// TwinCAT 3 PLC project Test_Projekt
// ProgramVersion: 3.1.4026.14
// libraries:
//   Tc2_Standard, * (Beckhoff Automation GmbH)
//   Tc2_System, * (Beckhoff Automation GmbH)
//   Tc2_Utilities, * (Beckhoff Automation GmbH)
//   Tc3_Module, * (Beckhoff Automation GmbH)
// project tree:
//   DUTs/Enums/ E_CAN_Object_Test_Error_Bits.TcDUT, E_Controlmode.TcDUT, E_Controlword_Bits.TcDUT, E_Homing_mode.TcDUT, E_LoggerState.TcDUT, E_Mode_of_operation.TcDUT, E_Test_step.TcDUT, E_Statemachine_State.TcDUT, E_Statemachine_Transition_Controlword.TcDUT, E_Statusword_Bits.TcDUT, E_SubElement_Types.TcDUT, J_E_Stop_Modes.TcDUT, J_E_Test_Ranking.TcDUT
//   DUTs/Structs/ ST_CAN_Object.TcDUT, ST_Homing_parameters.TcDUT, ST_Manufacturer_label.TcDUT, ST_Profile_velocity_parameters.TcDUT, ST_Statemachine_State.TcDUT, ST_Velocity_parameters.TcDUT
//   GVLs/ DS301_Object_List.TcGVL, DS302_Object_List.TcGVL, DS402_Object_List.TcGVL, GLB.TcGVL, Manufacturer_Label_Objects.TcGVL, Manufacturer_specific_Object_List.TcGVL, PDO.TcGVL
//   / PlcTask.TcTTO
//   POUs/ CAN_Object_Testing.TcPOU, Encoder_Alignment.TcPOU, Homing_Mode.TcPOU, J_Stop_Testing_SM.TcPOU, Velocity_Mode.TcPOU, MAIN.TcPOU, GET_STATE.TcPOU, Profile_Position_Mode.TcPOU, CONTROLWORD_STATE_CHANGE.TcPOU, Profile_Velocity_Mode.TcPOU, WRITE_Manufacturer_label.TcPOU, READ_Manufacturer_label.TcPOU
//   POUs/FB/Basic/ FB_NMT_WRITE.TcPOU, FB_SDO_READ.TcPOU, FB_SDO_READ_REAL.TcPOU, FB_SDO_WRITE.TcPOU, FB_SDO_WRITE_REAL.TcPOU
//   POUs/FB/ FB_DS402_Object_Testing.TcPOU, FB_Logger.TcPOU, FB_Object_List_Testing.TcPOU, FB_Object_Testing.TcPOU, FB_Sequenz_Testing.TcPOU
//   POUs/FUN/ DWORD_TO_BYTE_ARRAY.TcPOU, Get_Vel_RPM.TcPOU, J_Make_Message.TcPOU
// real-time tasks:
//   TASK PlcTask: cycle T#10ms, priority 20, ADS port 350
// I/O:
//   DEVICE Gerät 1 (EtherCAT), AmsNetId 5.156.6.243.2.1
//     Klemme 1 (EK1200) [EK1200-5000 EtherCAT Netzteil (2A E-Bus)]
//       Klemme 2 (EL1859) [EL1859 8K. Dig. Eingang 24V, 3ms, 8K. Dig. Ausgang 24V, 0.5A]
//       Klemme 3 (EL6751) [EL6751 CANopen Master]
//       Klemme 4 (EK1110) [EK1110 EtherCAT-Verlängerung]
//   DEVICE Gerät 3 (NOV-DP-RAM)
//   DEVICE Gerät 2 (EL6751), AmsNetId 5.156.6.243.3.1
//     Box 5 (CANopen Node)
// variable links:
//   Test_Projekt/Test_Projekt Instance <-> Device 1 (EtherCAT)/Term 1 (EK1200)/Term 2 (EL1859)
//     PlcTask Inputs/MAIN.bTaster{1..8} <-> Channel {1..8}/Input  (8 links)
//     PlcTask Outputs/MAIN.Stop_Testing_SM.OutputSTO1 <-> Channel 9/STO1
//     PlcTask Outputs/MAIN.Stop_Testing_SM.OutputSTO2 <-> Channel 10/STO2
//     PlcTask Outputs/MAIN.bLED{3..8} <-> Channel {11..16}/Output  (6 links)
//   Test_Projekt/Test_Projekt Instance <-> Device 2 (EL6751)/Box 5 (CANopen Node)
//     PlcTask Inputs/PDO.Current_actual_value <-> TxPDO 1/Inputs/Current_actual_value
//     PlcTask Inputs/PDO.DC_link_circuit_voltage <-> TxPDO 3/Inputs/DC link circuit voltage
//     PlcTask Inputs/PDO.Mode_of_operation_display <-> TxPDO 1/Inputs/Mode of operation display
//     PlcTask Inputs/PDO.Position_actual_value <-> TxPDO 2/Inputs/Position actual value
//     PlcTask Inputs/PDO.Statusword <-> TxPDO 1/Inputs/Statusword
//     PlcTask Inputs/PDO.Torque_actual_value <-> TxPDO 1/Inputs/Torque_actual_value
//     PlcTask Inputs/PDO.Velocity_actual_value <-> TxPDO 2/Inputs/Velocity_actual_value
//     PlcTask Inputs/PDO.vl_Velocity_actual_value <-> TxPDO 3/Inputs/Vl Velocity Actual Value
//     PlcTask Outputs/PDO.Controlword <-> RxPDO 1/Outputs/Controlword
//     PlcTask Outputs/PDO.Mode_of_operation <-> RxPDO 1/Outputs/Mode of operation
//     PlcTask Outputs/PDO.Profile_velocity <-> RxPDO 2/Outputs/Profile velocity
//     PlcTask Outputs/PDO.Target_position <-> RxPDO 3/Outputs/Target position
//     PlcTask Outputs/PDO.Target_torque <-> RxPDO 1/Outputs/Target_torque
//     PlcTask Outputs/PDO.Target_velocity <-> RxPDO 2/Outputs/Target velocity
//     PlcTask Outputs/PDO.vl_target_velocity <-> RxPDO 1/Outputs/vl_target_velocity

CONFIGURATION Test_Projekt
    RESOURCE PLC ON TwinCAT3
        TASK PlcTask(INTERVAL := T#10ms, PRIORITY := 20);
        PROGRAM MAIN WITH PlcTask : MAIN;
    END_RESOURCE
END_CONFIGURATION

// ---- DUTs/Enums/E_CAN_Object_Test_Error_Bits.TcDUT
{attribute 'qualified_only'}
{attribute 'strict'}
TYPE E_CAN_Object_Test_Error_Bits :
(
	No_error := 0
	
) WORD;
END_TYPE

// ---- DUTs/Enums/E_Controlmode.TcDUT
{attribute 'qualified_only'}
{attribute 'strict'}
TYPE E_Controlmode :
(
	IO_Testmode		:= 0,
	Manual			:= 1,
	Test_individual	:= 2,
	Test_sequence	:= 3	
) BYTE;
END_TYPE

// ---- DUTs/Enums/E_Controlword_Bits.TcDUT
{attribute 'qualified_only'}
{attribute 'strict'}
TYPE E_Controlword_Bits :
(
	Switch_on                   := 16#0001,
    Enable_voltage              := 16#0002,
    Quick_stop                  := 16#0004,   // Bit is low-active
    Enable_operation            := 16#0008,
    Operation_mode_specific_1   := 16#0010,
    Operation_mode_specific_2   := 16#0020,
    Operation_mode_specific_3   := 16#0040,
    Fault_reset                 := 16#0080,
    Halt                        := 16#0100,
    Operation_mode_specific_4   := 16#0200,
    Manufacturer_specific_1     := 16#0400,
    Manufacturer_specific_2     := 16#0800,
    Manufacturer_specific_3     := 16#1000,
    Manufacturer_specific_4     := 16#2000,
    Manufacturer_specific_5     := 16#4000,
    Manufacturer_specific_6     := 16#8000,
	
    // Profile position mode
    PPM_New_set_point           := Operation_mode_specific_1,
    PPM_Change_set_immediately  := Operation_mode_specific_2,
    PPM_Absolut_relative        := Operation_mode_specific_3,
    PPM_Change_on_setpoint      := Operation_mode_specific_4,

    // Velocity mode
    VM_Enable_ramp              := Operation_mode_specific_1,
    VM_Unlock_ramp              := Operation_mode_specific_2,
    VM_Reference_ramp           := Operation_mode_specific_3,

    // Profile velocity mode

    // Profile torque mode

    // Homing mode
    HM_Homing_operation_start   := Operation_mode_specific_1,

    // Interpolated position mode
    IPM_Enable_interpolation    := Operation_mode_specific_1

    // Cyclic synchronous position mode

    // Cyclic synchronous velocity mode

    // Cyclic synchronous torque mode

    // Cyclic synchronous torque mode with commutation angle

) WORD ;
END_TYPE

// ---- DUTs/Enums/E_Homing_mode.TcDUT
{attribute 'qualified_only'}
{attribute 'strict'}
TYPE E_Homing_mode :
(
	No_homing_methode_assigned			:= 0,
	
	
    Homing_on_current_position_obsolet 	:= 35,
    Homing_on_current_position 			:= 37
) SINT ;
END_TYPE

// ---- DUTs/Enums/E_LoggerState.TcDUT
{attribute 'qualified_only'}
{attribute 'strict'}
TYPE E_LoggerState :
(
	Open,
	Opening,
	Opening_Error,
	Opened,
	
	Writing,
	Writing_Error,
	
	Close,
	Closing,
	Closed,
	Closing_Error
) BYTE;
END_TYPE

// ---- DUTs/Enums/E_Mode_of_operation.TcDUT
{attribute 'qualified_only'}
{attribute 'strict'}
{attribute 'to_string'}
TYPE E_Mode_of_operation :
(
    No_mode_active                      := 0,
    Profile_position_mode               := 1,
    Velocity_mode                       := 2,
    Profile_velocity_mode               := 3,
    Profile_torque_mode                 := 4,
    Reserved                            := 5,
    Homing_mode                         := 6,
    Interpolated_position_mode          := 7,
    Cyclic_synchronous_position_mode    := 8,
    Cyclic_synchronous_velocity_mode    := 9,
    Cyclic_synchronous_torque_mode      := 10,
    Cyclic_synchronous_torque_mode_with_commutation_angle           := 11,
    Profile_position_mode_with_an_additional_feedback               := 12,
    Profile_velocity_mode_with_an_additional_feedback               := 13,
    Homing_mode_with_an_additional_feedback                         := 14,
    Cyclic_synchronous_position_mode_with_an_additional_feedback    := 15,
    Cyclic_synchronous_velocity_mode_with_an_additional_feedback    := 16,
	
	Phasing_mode						:= -121,
	Open_loop_voltage					:= -122,
	Non_commutated_current_mode			:= -123
) SINT ;
END_TYPE

// ---- DUTs/Enums/E_Test_step.TcDUT
{attribute 'qualified_only'}
{attribute 'strict'}
TYPE E_Test_step :
(
	// Change of state machine state
	Switch_on_disabled,		// Switch directly to state 'Switch on disabled' -> Set Controlword to 0
	Quick_stop_active,		// Switch directly to state 'Quick stop active' -> Set Controlword to 2
	Ready_to_switch_on,		// Switch directly to state 'Ready to switch on' -> Set Controlword to 6
	Switched_on,			// Switch directly to state 'Switched on' -> Set Controlword to 7
	Operation_enabled,		// Switch directly to state 'Operation enabled' -> Set Controlword to F
	
	// Change of Mode of Operation
	No_Mode,				// Set Mode of Operation to 'No mode'
	Mode_PPM,				// Set Mode of Operation to 'Profile Position Mode'
	Mode_VM,				// Set Mode of Operation to 'Velocity Mode'
	Mode_PVM,				// Set Mode of Operation to 'Profile Velocity Mode'
	Mode_PTM,				// Set Mode of Operation to 'Profile Torque Mode'
	Mode_HM,				// Set Mode of Operation to 'Homing Mode'
	Mode_IPM,				// Set Mode of Operation to 'Interpolated Position Mode'
	
	// Init values
	Factor_group_rpm,		// Set the factor group to use rpm as user-defined velocity unit
	
	// Setting values
	Velocity_window_30rpm,	// Set 'Velocity_window' to value 30
	Velocity_window_100ms,	// Set 'Velocity window time' to value 100
	Acceleration_1000,		// Set 'Profile acceleration' to value 1000
	Deceleration_1000,		// Set 'Profile deceleration' to value 1000
	PPM_Velocity_1000,		// Set 'Profile velocity' to value 1000
	PVM_Velocity_1000,		// Set 'Target velocity' to value 1000
		
	// Check conditions
	Check_Statusword_Target_reached_200ms,	// Check if the Statusword 'Target reached' bit is set within 200 ms 
	
	// Waiting times
	Wait_10ms,				// Wait 10 ms 	(= 1 cycle)
	Wait_50ms,				// Wait 50 ms 	(= 5 cycle)
	Wait_100ms,				// Wait 100 ms 	(= 10 cycle)
	Wait_250ms,				// Wait 250 ms 	(= 25 cycle)
	Wait_500ms,				// Wait 500 ms 	(= 50 cycle)
	Wait_1000ms,			// Wait 1 s 	(= 100 cycle)
	Wait_2500ms				// Wait 2,5 s 	(= 250 cycle)
		
) BYTE;
END_TYPE

// ---- DUTs/Enums/E_Statemachine_State.TcDUT
{attribute 'qualified_only'}
{attribute 'strict'}
TYPE E_Statemachine_State :
(
    Not_ready_to_switch_on  := 0,
    Switch_on_disabled      := 1,
    Ready_to_switch_on      := 2,
    Switched_on             := 3,
    Operation_enabled       := 4,
    Quick_stop_active       := 5,
    Fault_reaction_active   := 6,
    Fault                   := 7,

    unknown                 := 255
) BYTE ;
END_TYPE

// ---- DUTs/Enums/E_Statemachine_Transition_Controlword.TcDUT
{attribute 'qualified_only'}
{attribute 'strict'}
TYPE E_Statemachine_Transition_Controlword :
(
    Switch_on_disabled	:= 16#0000,
    Ready_to_switch_on	:= 16#0006,
    Switched_on			:= 16#0007,
    Operation_enabled	:= 16#000F,
    Quick_stop_active	:= 16#0002,
    Faultreset_step_1	:= 16#0000,
    Faultreset_step_2	:= 16#0080
) WORD ;
END_TYPE

// ---- DUTs/Enums/E_Statusword_Bits.TcDUT
{attribute 'qualified_only'}
{attribute 'strict'}
TYPE E_Statusword_Bits :
(
    Ready_to_switch_on          := 16#0001,
    Switched_on                 := 16#0002,
    Operation_enabled           := 16#0004,
    Fault                       := 16#0008,
    Voltage_enabled             := 16#0010,
    Quick_stop                  := 16#0020,   // Bit is low-active
    Switch_on_disabled          := 16#0040,
    Warning                     := 16#0080,
    Manufacturer_specific_1     := 16#0100,
    Remote                      := 16#0200,
    Target_reached              := 16#0400,
    Internal_limit_active       := 16#0800,
    Operation_mode_specific_1   := 16#1000,
    Operation_mode_specific_2   := 16#2000,
    Manufacturer_specific_2     := 16#4000,
    Manufacturer_specific_3     := 16#8000,

    // Profile position mode
    PPM_Set_point_acknowledge   := Operation_mode_specific_1,
    PPM_Following_error         := Operation_mode_specific_2,

    // Velocity mode

    // Profile velocity mode
    PVM_Speed                   := Operation_mode_specific_1,
    PVM_Max_slippage_error      := Operation_mode_specific_2,

    // Profile torque mode

    // Homing mode
    HM_Homing_attained          := Operation_mode_specific_1,
    HM_Homing_error             := Operation_mode_specific_2,

    // Interpolated position mode
    IPM_IP_mode_active          := Operation_mode_specific_1,
    IPM_Following_error         := Operation_mode_specific_2,

    // Cyclic synchronous position mode
    CSPM_Drive_follows_the_command_value    := Operation_mode_specific_1,
    CSPM_Following_error                    := Operation_mode_specific_2,

    // Cyclic synchronous velocity mode
    CSVM_Drive_follows_the_command_value    := Operation_mode_specific_1,

    // Cyclic synchronous torque mode
    CSTM_Drive_follows_the_command_value    := Operation_mode_specific_1,

    // Cyclic synchronous torque mode with commutation angle
    CSTCAM_Drive_follows_the_command_value  := Operation_mode_specific_1
) WORD ;
END_TYPE

// ---- DUTs/Enums/E_SubElement_Types.TcDUT
{attribute 'qualified_only'}
{attribute 'strict'}
TYPE E_SubElement_Types :
(
	No 						:= 0,
	
	With_fix_subelements	:= 1,
	With_list 				:= 2,
	
	Fix_subelement			:= 17,	
	List_element			:= 18
) BYTE;
END_TYPE

// ---- DUTs/Enums/J_E_Stop_Modes.TcDUT
{attribute 'qualified_only'}
{attribute 'strict'}
{attribute 'to_string'}
TYPE J_E_Stop_Modes :
(
		Switch_On,					//schnell runterrampen -> Switched on
		Shutdown,					//Disable PS
		Switch_On_Disabled,			//Disable PS
		Vel_To_Zero,				//stillstand mit dehmoment 
		Halt,						//stillstand mit dehmoment -> Weiterdrehen
		Quick_Stop,					//schnell runterrampen -> Switch on Disabled
		STO1,						//Disable PS
		STO2,						//Disable PS
		Fault						//DISABLE PS
);
END_TYPE

// ---- DUTs/Enums/J_E_Test_Ranking.TcDUT
{attribute 'qualified_only'}
{attribute 'strict'}
{attribute 'to_string'}
TYPE J_E_Test_Ranking :
(
	OK := 0,
	Not_OK := 1,
	Issues := 2
);
END_TYPE

// ---- DUTs/Structs/ST_CAN_Object.TcDUT
TYPE ST_CAN_Object :
STRUCT
	Name				: STRING(80);
	Index				: WORD := 0;
	Subindex			: BYTE := 0;
	
	Length_Tested		: BOOL := FALSE;	// Test is performed
	Length_Error		: DWORD:= 0;		// Error number
	Length_Target		: BYTE := 4;		// Target value (must be set at test)
	Length				: BYTE := 4;
		
	Readable_Tested		: BOOL := FALSE;	// Test is performed
	Readable_Error		: DWORD:= 0;		// Error number
	Readable_Target		: BOOL := TRUE;		// Target value (must be set at test)
	Readable			: BOOL := TRUE;
	
	Writable_Tested		: BOOL := FALSE;	// Test is performed
	Writable_Error		: DWORD:= 0;		// Error number
	Writable_Target		: BOOL := TRUE;		// Target value (must be set at test)
	Writable			: BOOL := TRUE;
	
	TPDO_Mappable_Tested: BOOL := FALSE;	// Test is performed
	TPDO_Mappable_Error	: DWORD:= 0;		// Error number
	TPDO_Mappable_Target: BOOL := FALSE;	// Target value (must be set at test)
	TPDO_Mappable		: BOOL := FALSE;
	
	RPDO_Mappable_Tested: BOOL := FALSE;	// Test is performed
	RPDO_Mappable_Error	: DWORD:= 0;		// Error number
	RPDO_Mappable_Target: BOOL := FALSE;	// Target value (must be set at test)
	RPDO_Mappable		: BOOL := FALSE;
	
	Error				: BOOL	:=FALSE;	// Has an error occurred in at least one test?
	
	Read_Value			: DWORD := 0;
	Write_Value			: DWORD := 0;
	Write_Value_Usage	: BOOL := FALSE;	// Which value should be used for the Writable test? True: Write_Value / False: Read_Value (in case the object is not readable '0' is used)
	
	Default_Value		: DWORD := 0;
	
	Mandatory			: BYTE := 0;
	SubElements			: E_SubElement_types := E_SubElement_types.No;
END_STRUCT
END_TYPE

// ---- DUTs/Structs/ST_Homing_parameters.TcDUT
TYPE ST_Homing_parameters :
STRUCT
	Homing_mode		: E_Homing_mode;		// 0x6098, 0, 8 bit
	Speed_switch	: DWORD;				// 0x6099, 1, 32 bit
	Speed_zero		: DWORD;				// 0x6099, 2, 32 bit
	Acceleration	: DWORD;				// 0x609A, 0, 32 bit
END_STRUCT
END_TYPE

// ---- DUTs/Structs/ST_Manufacturer_label.TcDUT
TYPE ST_Manufacturer_label :
STRUCT
	Serial_Number			: DWORD;
	Min_v					: DWORD;
	Max_v					: DWORD;
	Motor_rated_current		: DWORD;
	Drive_rated_current		: DWORD;
	Max_current				: WORD;
	Motor_rated_torque		: DWORD;
	Max_torque				: WORD;
	Motor_rated_speed		: DWORD;
	Number_of_pole_pairs	: WORD;
	Motor_torque_constant	: REAL;
	Flux_producing_P_gain	: REAL;
	Flux_producing_I_gain	: REAL;
	Torque_producing_P_gain	: REAL;
	Torque_producing_I_gain	: REAL;
	Magnetic_encoder_offset	: WORD;
	Motor_with_brake		: WORD;
	Encoder_mode_adjust		: WORD;
	Motor_max_speed			: WORD;
	Rotor_inertia			: REAL;
	Motor_time_at_peak		: REAL;
	Drive_time_at_peak		: REAL;
	Singleturn_resolution	: BYTE;
	Multiturn_resolution	: BYTE;	
END_STRUCT
END_TYPE

// ---- DUTs/Structs/ST_Profile_velocity_parameters.TcDUT
TYPE ST_Profile_velocity_parameters :
STRUCT
	Target_velocity			: DINT;		// 0x60FF, 0, 32 bit
	Profile_acceleration	: DWORD;	// 0x6083, 0, 32 bit
	Profile_deceleration	: DWORD;	// 0x6084, 0, 32 bit
END_STRUCT
END_TYPE

// ---- DUTs/Structs/ST_Statemachine_State.TcDUT
TYPE ST_Statemachine_State :
STRUCT
	State			: E_Statemachine_State;
    Name			: STRING(25);
    Statusword		: E_Statemachine_Statusword;
	Statusword_mask	: E_Statemachine_Statusword_Mask;
	Statemachine_Transition_Controlword	: E_Statemachine_Transition_Controlword;
END_STRUCT
END_TYPE

// ---- DUTs/Structs/ST_Velocity_parameters.TcDUT
TYPE ST_Velocity_parameters :
STRUCT
	vl_target_velocity			: INT;		// 0x6042, 0, 16 bit
	vl_velocity_acceleration	: DWORD;	// 0x6048, 0, 32 bit
	vl_velocity_deceleration	: DWORD;	// 0x6049, 0, 32 bit
END_STRUCT
END_TYPE

// ---- GVLs/DS301_Object_List.TcGVL
{attribute 'qualified_only'}
VAR_GLOBAL
	Device_type															: ST_CAN_Object := (Name:='Device type', 														Index:=16#1000, 			 			Writable:=FALSE);
	Error_register														: ST_CAN_Object := (Name:='Error register', 													Index:=16#1001, 			 Length:=1, Writable:=FALSE);
	Manufacturer_status_register										: ST_CAN_Object := (Name:='Manufacturer status register', 										Index:=16#1002, 			 			Writable:=FALSE);
	Pre_defined_error_field_Number_of_errors							: ST_CAN_Object := (Name:='Pre-defined error field_Number of errors',							Index:=16#1003, 			 Length:=1, 										SubElements:=E_SubElement_types.With_list);
	Pre_defined_error_field_Standard_error_field_1						: ST_CAN_Object := (Name:='Pre-defined error field_Standard error field 1',						Index:=16#1003, Subindex:=1, 			Writable:=FALSE,						SubElements:=E_SubElement_types.List_element);
	COB_ID_SYNC															: ST_CAN_Object := (Name:='COB-ID SYNC',														Index:=16#1005, 			 			Writable:=FALSE, Default_Value:=16#80);
	Communication_cycle_period											: ST_CAN_Object := (Name:='Communication cycle period',											Index:=16#1006);
	Synchronous_window_length											: ST_CAN_Object := (Name:='Synchronous window length',											Index:=16#1007);
	Manufacturer_device_name											: ST_CAN_Object := (Name:='Manufacturer device name', 											Index:=16#1008, 			 Length:=0, Writable:=FALSE);
	Manufacturer_hardware_version										: ST_CAN_Object := (Name:='Manufacturer hardware version',										Index:=16#1009, 			 Length:=0, Writable:=FALSE);
	Manufacturer_software_version										: ST_CAN_Object := (Name:='Manufacturer software version',										Index:=16#100A, 			 Length:=0, Writable:=FALSE);
	Guard_time															: ST_CAN_Object := (Name:='Guard time', 														Index:=16#100C, 			 Length:=2, Writable:=FALSE);
	Life_time_factor													: ST_CAN_Object := (Name:='Life time factor', 													Index:=16#100D, 			 Length:=1, Writable:=FALSE);
	store_parameters_highest_sub_index_supported						: ST_CAN_Object := (Name:='store parameters_highest sub-index supported', 						Index:=16#1010, 			 Length:=1, Writable:=FALSE, Default_Value:=4, 		SubElements:=E_SubElement_types.With_fix_subelements);
	store_parameters_save_all_parameters								: ST_CAN_Object := (Name:='store parameters_save all parameters', 								Index:=16#1010, Subindex:=1, 													SubElements:=E_SubElement_types.Fix_subelement);
	store_parameters_save_communication_parameters						: ST_CAN_Object := (Name:='store parameters_save communication parameters', 					Index:=16#1010, Subindex:=2, 													SubElements:=E_SubElement_types.Fix_subelement);
	store_parameters_save_application_parameters						: ST_CAN_Object := (Name:='store parameters_save application parameters', 						Index:=16#1010, Subindex:=3, 													SubElements:=E_SubElement_types.Fix_subelement);
	store_parameters_save_manufacture_label								: ST_CAN_Object := (Name:='store parameters_save manufacture label', 							Index:=16#1010, Subindex:=4, 													SubElements:=E_SubElement_types.Fix_subelement);
	restore_default_parameters_highest_sub_index_supported				: ST_CAN_Object := (Name:='restore default parameters_highest sub-index supported', 			Index:=16#1011, 			 Length:=1, Writable:=FALSE, Default_Value:=4, 		SubElements:=E_SubElement_types.With_fix_subelements);
	restore_default_parameters_restore_all_default_parameters			: ST_CAN_Object := (Name:='restore default parameters_restore all default parameters', 			Index:=16#1011, Subindex:=1,													SubElements:=E_SubElement_types.Fix_subelement);
	restore_default_parameters_restore_communication_default_parameters	: ST_CAN_Object := (Name:='restore default parameters_restore communication default parameters',Index:=16#1011, Subindex:=2,													SubElements:=E_SubElement_types.Fix_subelement);
	restore_default_parameters_restore_application_default_parameters	: ST_CAN_Object := (Name:='restore default parameters_restore application default parameters', 	Index:=16#1011, Subindex:=3,													SubElements:=E_SubElement_types.Fix_subelement);
	restore_default_parameters_restore_default_manufacture_label		: ST_CAN_Object := (Name:='restore default parameters_restore default manufacture label', 		Index:=16#1011, Subindex:=4,													SubElements:=E_SubElement_types.Fix_subelement);
	COB_ID_time_stamp_message											: ST_CAN_Object := (Name:='COB-ID time stamp message', 											Index:=16#1012);
	High_resolution_time_stamp											: ST_CAN_Object := (Name:='High resolution time stamp', 										Index:=16#1013);
	COB_ID_emergency_message											: ST_CAN_Object := (Name:='COB-ID emergency message', 											Index:=16#1014);
	Inhibit_time_emergency_message										: ST_CAN_Object := (Name:='Inhibit time emergency message', 									Index:=16#1015, 			 Length:=2);
	Consumer_heartbeat_time_highest_sub_index_supported					: ST_CAN_Object := (Name:='Consumer heartbeat time_highest sub-index supported', 				Index:=16#1016, 			 Length:=1, 										SubElements:=E_SubElement_types.With_list);
	Consumer_heartbeat_time_1											: ST_CAN_Object := (Name:='Consumer heartbeat time 1',											Index:=16#1016, Subindex:=1, 													SubElements:=E_SubElement_types.List_element);
	Producer_heartbeat_time												: ST_CAN_Object := (Name:='Producer heartbeat time', 											Index:=16#1017, 			 Length:=2);
	Identity_object_Highest_sub_index_supported							: ST_CAN_Object := (Name:='Identity object_Highest sub-index supported', 						Index:=16#1018, 			 Length:=1, Writable:=FALSE, Default_Value:=4, 		SubElements:=E_SubElement_types.With_fix_subelements);
	Identity_object_Vendor_ID											: ST_CAN_Object := (Name:='Identity object_Vendor-ID', 											Index:=16#1018, Subindex:=1, 			Writable:=FALSE, 					 	SubElements:=E_SubElement_types.Fix_subelement);
	Identity_object_Product_code										: ST_CAN_Object := (Name:='Identity object_Product code',										Index:=16#1018, Subindex:=2, 			Writable:=FALSE, 					 	SubElements:=E_SubElement_types.Fix_subelement);
	Identity_object_Revision_number										: ST_CAN_Object := (Name:='Identity object_Revision number',									Index:=16#1018, Subindex:=3, 			Writable:=FALSE, 					 	SubElements:=E_SubElement_types.Fix_subelement);
	Identity_object_Serial_number										: ST_CAN_Object := (Name:='Identity object_Serial number',										Index:=16#1018, Subindex:=4, 			Writable:=FALSE, 					 	SubElements:=E_SubElement_types.Fix_subelement);	
	Synchronous_counter_overflow_value									: ST_CAN_Object := (Name:='Synchronous counter overflow value', 								Index:=16#1019, 			 Length:=1);
	Verify_configuration_highest_sub_index_supported					: ST_CAN_Object := (Name:='Verify configuration_Highest sub-index supported', 					Index:=16#1020, 			 Length:=1, Writable:=FALSE, Default_Value:=2, 		SubElements:=E_SubElement_types.With_fix_subelements);
	Verify_configuration_Configuration_date								: ST_CAN_Object := (Name:='Verify configuration_Configuration date', 							Index:=16#1020, Subindex:=1, 													SubElements:=E_SubElement_types.Fix_subelement);
	Verify_configuration_Configuration_time								: ST_CAN_Object := (Name:='Verify configuration_Configuration time', 							Index:=16#1020, Subindex:=2, 													SubElements:=E_SubElement_types.Fix_subelement);

	// SDO setting
	Server_SDO_Parameter_0_Number_of_entries							: ST_CAN_Object := (Name:='Server SDO Parameter 0_Number of entries', 							Index:=16#1200, 			 Length:=1, Writable:=FALSE, Default_Value:=2, 		SubElements:=E_SubElement_types.With_fix_subelements);
	Server_SDO_Parameter_0_COB_ID_Client_to_Server						: ST_CAN_Object := (Name:='Server SDO Parameter 0_COB ID Client to Server', 					Index:=16#1200, Subindex:=1, 			Writable:=FALSE,						SubElements:=E_SubElement_types.Fix_subelement);
	Server_SDO_Parameter_0_COB_ID_Server_to_Client						: ST_CAN_Object := (Name:='Server SDO Parameter 0_COB ID Server to Client', 					Index:=16#1200, Subindex:=2, 			Writable:=FALSE,						SubElements:=E_SubElement_types.Fix_subelement);
	
	// PDO setting
	RPDO1_communication_parameter_Highest_sub_index_supported			: ST_CAN_Object := (Name:='RPDO communication parameter_Highest sub-index supported', 			Index:=16#1400, 			 Length:=1, Writable:=FALSE, Default_Value:=5,		SubElements:=E_SubElement_types.With_fix_subelements);
	RPDO1_communication_parameter_COB_ID_used_by_RPDO					: ST_CAN_Object := (Name:='RPDO communication parameter_COB-ID used by RPDO', 					Index:=16#1400, Subindex:=1,													SubElements:=E_SubElement_types.Fix_subelement);
	RPDO1_communication_parameter_Transmission_type						: ST_CAN_Object := (Name:='RPDO communication parameter_Transmission type', 					Index:=16#1400, Subindex:=2, Length:=1, 										SubElements:=E_SubElement_types.Fix_subelement);
	RPDO1_communication_parameter_Event_timer							: ST_CAN_Object := (Name:='RPDO communication parameter_Event timer', 							Index:=16#1400, Subindex:=5, Length:=2, 										SubElements:=E_SubElement_types.Fix_subelement);
	RPDO2_communication_parameter_Highest_sub_index_supported			: ST_CAN_Object := (Name:='RPDO communication parameter_Highest sub-index supported',			Index:=16#1401, 			 Length:=1, Writable:=FALSE, Default_Value:=5, 		SubElements:=E_SubElement_types.With_fix_subelements);
	RPDO2_communication_parameter_COB_ID_used_by_RPDO					: ST_CAN_Object := (Name:='RPDO communication parameter_COB-ID used by RPDO', 					Index:=16#1401, Subindex:=1,													SubElements:=E_SubElement_types.Fix_subelement);
	RPDO2_communication_parameter_Transmission_type						: ST_CAN_Object := (Name:='RPDO communication parameter_Transmission type', 					Index:=16#1401, Subindex:=2, Length:=1, 										SubElements:=E_SubElement_types.Fix_subelement);
	RPDO2_communication_parameter_Event_timer							: ST_CAN_Object := (Name:='RPDO communication parameter_Event timer', 							Index:=16#1401, Subindex:=5, Length:=2,											SubElements:=E_SubElement_types.Fix_subelement);
	RPDO3_communication_parameter_Highest_sub_index_supported			: ST_CAN_Object := (Name:='RPDO communication parameter_Highest sub-index supported', 			Index:=16#1402, 			 Length:=1, Writable:=FALSE, Default_Value:=5, 		SubElements:=E_SubElement_types.With_fix_subelements);
	RPDO3_communication_parameter_COB_ID_used_by_RPDO					: ST_CAN_Object := (Name:='RPDO communication parameter_COB-ID used by RPDO', 					Index:=16#1402, Subindex:=1,													SubElements:=E_SubElement_types.Fix_subelement);
	RPDO3_communication_parameter_Transmission_type						: ST_CAN_Object := (Name:='RPDO communication parameter_Transmission type', 					Index:=16#1402, Subindex:=2, Length:=1, 										SubElements:=E_SubElement_types.Fix_subelement);
	RPDO3_communication_parameter_Event_timer							: ST_CAN_Object := (Name:='RPDO communication parameter_Event timer', 							Index:=16#1402, Subindex:=5, Length:=2,											SubElements:=E_SubElement_types.Fix_subelement);
	RPDO4_communication_parameter_Highest_sub_index_supported			: ST_CAN_Object := (Name:='RPDO communication parameter_Highest sub-index supported', 			Index:=16#1403, 			 Length:=1, Writable:=FALSE, Default_Value:=5,		SubElements:=E_SubElement_types.With_fix_subelements);
	RPDO4_communication_parameter_COB_ID_used_by_RPDO					: ST_CAN_Object := (Name:='RPDO communication parameter_COB-ID used by RPDO', 					Index:=16#1403, Subindex:=1,													SubElements:=E_SubElement_types.Fix_subelement);
	RPDO4_communication_parameter_Transmission_type						: ST_CAN_Object := (Name:='RPDO communication parameter_Transmission type', 					Index:=16#1403, Subindex:=2, Length:=1, 										SubElements:=E_SubElement_types.Fix_subelement);
	RPDO4_communication_parameter_Event_timer							: ST_CAN_Object := (Name:='RPDO communication parameter_Event timer', 							Index:=16#1403, Subindex:=5, Length:=2,											SubElements:=E_SubElement_types.Fix_subelement);
	RPDO1_mapping_parameter_Number_of_mapped_application_objects_in_PDO	: ST_CAN_Object := (Name:='RPDO mapping parameter_Number of mapped application objects in PDO', Index:=16#1600, 			 Length:=1, 										SubElements:=E_SubElement_types.With_fix_subelements);
	RPDO1_mapping_parameter_Application_object_1						: ST_CAN_Object := (Name:='RPDO mapping parameter_Application object 1', 						Index:=16#1600, Subindex:=1, 													SubElements:=E_SubElement_types.Fix_subelement);
	RPDO1_mapping_parameter_Application_object_2						: ST_CAN_Object := (Name:='RPDO mapping parameter_Application object 2', 						Index:=16#1600, Subindex:=2, 													SubElements:=E_SubElement_types.Fix_subelement);
	RPDO1_mapping_parameter_Application_object_3						: ST_CAN_Object := (Name:='RPDO mapping parameter_Application object 3', 						Index:=16#1600, Subindex:=3, 													SubElements:=E_SubElement_types.Fix_subelement);
	RPDO1_mapping_parameter_Application_object_4						: ST_CAN_Object := (Name:='RPDO mapping parameter_Application object 4', 						Index:=16#1600, Subindex:=4, 													SubElements:=E_SubElement_types.Fix_subelement);
	RPDO1_mapping_parameter_Application_object_5						: ST_CAN_Object := (Name:='RPDO mapping parameter_Application object 5', 						Index:=16#1600, Subindex:=5, 													SubElements:=E_SubElement_types.Fix_subelement);
	RPDO1_mapping_parameter_Application_object_6						: ST_CAN_Object := (Name:='RPDO mapping parameter_Application object 6',						Index:=16#1600, Subindex:=6, 													SubElements:=E_SubElement_types.Fix_subelement);
	RPDO1_mapping_parameter_Application_object_7						: ST_CAN_Object := (Name:='RPDO mapping parameter_Application object 7',						Index:=16#1600, Subindex:=7, 													SubElements:=E_SubElement_types.Fix_subelement);
	RPDO1_mapping_parameter_Application_object_8						: ST_CAN_Object := (Name:='RPDO mapping parameter_Application object 8', 						Index:=16#1600, Subindex:=8, 													SubElements:=E_SubElement_types.Fix_subelement);
	RPDO2_mapping_parameter_Number_of_mapped_application_objects_in_PDO	: ST_CAN_Object := (Name:='RPDO mapping parameter_Number of mapped application objects in PDO', Index:=16#1601, 			 Length:=1, 										SubElements:=E_SubElement_types.With_fix_subelements);
	RPDO2_mapping_parameter_Application_object_1						: ST_CAN_Object := (Name:='RPDO mapping parameter_Application object 1', 						Index:=16#1601, Subindex:=1, 													SubElements:=E_SubElement_types.Fix_subelement);
	RPDO2_mapping_parameter_Application_object_2						: ST_CAN_Object := (Name:='RPDO mapping parameter_Application object 2', 						Index:=16#1601, Subindex:=2, 													SubElements:=E_SubElement_types.Fix_subelement);
	RPDO2_mapping_parameter_Application_object_3						: ST_CAN_Object := (Name:='RPDO mapping parameter_Application object 3', 						Index:=16#1601, Subindex:=3, 													SubElements:=E_SubElement_types.Fix_subelement);
	RPDO2_mapping_parameter_Application_object_4						: ST_CAN_Object := (Name:='RPDO mapping parameter_Application object 4', 						Index:=16#1601, Subindex:=4, 													SubElements:=E_SubElement_types.Fix_subelement);
	RPDO2_mapping_parameter_Application_object_5						: ST_CAN_Object := (Name:='RPDO mapping parameter_Application object 5', 						Index:=16#1601, Subindex:=5, 													SubElements:=E_SubElement_types.Fix_subelement);
	RPDO2_mapping_parameter_Application_object_6						: ST_CAN_Object := (Name:='RPDO mapping parameter_Application object 6', 						Index:=16#1601, Subindex:=6, 													SubElements:=E_SubElement_types.Fix_subelement);
	RPDO2_mapping_parameter_Application_object_7						: ST_CAN_Object := (Name:='RPDO mapping parameter_Application object 7', 						Index:=16#1601, Subindex:=7, 													SubElements:=E_SubElement_types.Fix_subelement);
	RPDO2_mapping_parameter_Application_object_8						: ST_CAN_Object := (Name:='RPDO mapping parameter_Application object 8', 						Index:=16#1601, Subindex:=8, 													SubElements:=E_SubElement_types.Fix_subelement);
	RPDO3_mapping_parameter_Number_of_mapped_application_objects_in_PDO	: ST_CAN_Object := (Name:='RPDO mapping parameter_Number of mapped application objects in PDO', Index:=16#1602, 			 Length:=1, 										SubElements:=E_SubElement_types.With_fix_subelements);
	RPDO3_mapping_parameter_Application_object_1						: ST_CAN_Object := (Name:='RPDO mapping parameter_Application object 1', 						Index:=16#1602, Subindex:=1, 													SubElements:=E_SubElement_types.Fix_subelement);
	RPDO3_mapping_parameter_Application_object_2						: ST_CAN_Object := (Name:='RPDO mapping parameter_Application object 2', 						Index:=16#1602, Subindex:=2, 													SubElements:=E_SubElement_types.Fix_subelement);
	RPDO3_mapping_parameter_Application_object_3						: ST_CAN_Object := (Name:='RPDO mapping parameter_Application object 3', 						Index:=16#1602, Subindex:=3, 													SubElements:=E_SubElement_types.Fix_subelement);
	RPDO3_mapping_parameter_Application_object_4						: ST_CAN_Object := (Name:='RPDO mapping parameter_Application object 4', 						Index:=16#1602, Subindex:=4, 													SubElements:=E_SubElement_types.Fix_subelement);
	RPDO3_mapping_parameter_Application_object_5						: ST_CAN_Object := (Name:='RPDO mapping parameter_Application object 5', 						Index:=16#1602, Subindex:=5, 													SubElements:=E_SubElement_types.Fix_subelement);
	RPDO3_mapping_parameter_Application_object_6						: ST_CAN_Object := (Name:='RPDO mapping parameter_Application object 6', 						Index:=16#1602, Subindex:=6, 													SubElements:=E_SubElement_types.Fix_subelement);
	RPDO3_mapping_parameter_Application_object_7						: ST_CAN_Object := (Name:='RPDO mapping parameter_Application object 7', 						Index:=16#1602, Subindex:=7, 													SubElements:=E_SubElement_types.Fix_subelement);
	RPDO3_mapping_parameter_Application_object_8						: ST_CAN_Object := (Name:='RPDO mapping parameter_Application object 8', 						Index:=16#1602, Subindex:=8, 													SubElements:=E_SubElement_types.Fix_subelement);
	RPDO4_mapping_parameter_Number_of_mapped_application_objects_in_PDO	: ST_CAN_Object := (Name:='RPDO mapping parameter_Number of mapped application objects in PDO', Index:=16#1603, 			 Length:=1, 										SubElements:=E_SubElement_types.With_fix_subelements);
	RPDO4_mapping_parameter_Application_object_1						: ST_CAN_Object := (Name:='RPDO mapping parameter_Application object 1', 						Index:=16#1603, Subindex:=1, 													SubElements:=E_SubElement_types.Fix_subelement);
	RPDO4_mapping_parameter_Application_object_2						: ST_CAN_Object := (Name:='RPDO mapping parameter_Application object 2', 						Index:=16#1603, Subindex:=2, 													SubElements:=E_SubElement_types.Fix_subelement);
	RPDO4_mapping_parameter_Application_object_3						: ST_CAN_Object := (Name:='RPDO mapping parameter_Application object 3', 						Index:=16#1603, Subindex:=3, 													SubElements:=E_SubElement_types.Fix_subelement);
	RPDO4_mapping_parameter_Application_object_4						: ST_CAN_Object := (Name:='RPDO mapping parameter_Application object 4', 						Index:=16#1603, Subindex:=4, 													SubElements:=E_SubElement_types.Fix_subelement);
	RPDO4_mapping_parameter_Application_object_5						: ST_CAN_Object := (Name:='RPDO mapping parameter_Application object 5', 						Index:=16#1603, Subindex:=5, 													SubElements:=E_SubElement_types.Fix_subelement);
	RPDO4_mapping_parameter_Application_object_6						: ST_CAN_Object := (Name:='RPDO mapping parameter_Application object 6', 						Index:=16#1603, Subindex:=6, 													SubElements:=E_SubElement_types.Fix_subelement);
	RPDO4_mapping_parameter_Application_object_7						: ST_CAN_Object := (Name:='RPDO mapping parameter_Application object 7', 						Index:=16#1603, Subindex:=7, 													SubElements:=E_SubElement_types.Fix_subelement);
	RPDO4_mapping_parameter_Application_object_8						: ST_CAN_Object := (Name:='RPDO mapping parameter_Application object 8', 						Index:=16#1603, Subindex:=8, 													SubElements:=E_SubElement_types.Fix_subelement);
	TPDO1_communication_parameter_Highest_sub_index_supported			: ST_CAN_Object := (Name:='TPDO communication parameter_Highest sub-index supported', 			Index:=16#1800, 			 Length:=1, Writable:=FALSE, Default_Value:=6, 		SubElements:=E_SubElement_types.With_fix_subelements);
	TPDO1_communication_parameter_COB_ID_used_by_TPDO					: ST_CAN_Object := (Name:='TPDO communication parameter_COB-ID used by TPDO', 					Index:=16#1800, Subindex:=1, 													SubElements:=E_SubElement_types.Fix_subelement);
	TPDO1_communication_parameter_Transmission_type						: ST_CAN_Object := (Name:='TPDO communication parameter_Transmission type', 					Index:=16#1800, Subindex:=2, Length:=1, 										SubElements:=E_SubElement_types.Fix_subelement);
	TPDO1_communication_parameter_Inhibit_time							: ST_CAN_Object := (Name:='TPDO communication parameter_Inhibit time', 							Index:=16#1800, Subindex:=3, Length:=2, 										SubElements:=E_SubElement_types.Fix_subelement);
	TPDO1_communication_parameter_Event_timer							: ST_CAN_Object := (Name:='TPDO communication parameter_Event timer', 							Index:=16#1800, Subindex:=5, Length:=2, 										SubElements:=E_SubElement_types.Fix_subelement);
	TPDO1_communication_parameter_SYNC_start_value						: ST_CAN_Object := (Name:='TPDO communication parameter_SYNC start value', 						Index:=16#1800, Subindex:=6, Length:=1, 										SubElements:=E_SubElement_types.Fix_subelement);	
	TPDO2_communication_parameter_Highest_sub_index_supported			: ST_CAN_Object := (Name:='TPDO communication parameter_Highest sub-index supported', 			Index:=16#1801, 			 Length:=1, Writable:=FALSE, Default_Value:=6, 		SubElements:=E_SubElement_types.With_fix_subelements);
	TPDO2_communication_parameter_COB_ID_used_by_TPDO					: ST_CAN_Object := (Name:='TPDO communication parameter_COB-ID used by TPDO', 					Index:=16#1801, Subindex:=1, 													SubElements:=E_SubElement_types.Fix_subelement);
	TPDO2_communication_parameter_Transmission_type						: ST_CAN_Object := (Name:='TPDO communication parameter_Transmission type', 					Index:=16#1801, Subindex:=2, Length:=1, 										SubElements:=E_SubElement_types.Fix_subelement);
	TPDO2_communication_parameter_Inhibit_time							: ST_CAN_Object := (Name:='TPDO communication parameter_Inhibit time', 							Index:=16#1801, Subindex:=3, Length:=2, 										SubElements:=E_SubElement_types.Fix_subelement);
	TPDO2_communication_parameter_Event_timer							: ST_CAN_Object := (Name:='TPDO communication parameter_Event timer', 							Index:=16#1801, Subindex:=5, Length:=2, 										SubElements:=E_SubElement_types.Fix_subelement);
	TPDO2_communication_parameter_SYNC_start_value						: ST_CAN_Object := (Name:='TPDO communication parameter_SYNC start value', 						Index:=16#1801, Subindex:=6, Length:=1, 										SubElements:=E_SubElement_types.Fix_subelement);
	TPDO3_communication_parameter_Highest_sub_index_supported			: ST_CAN_Object := (Name:='TPDO communication parameter_Highest sub-index supported', 			Index:=16#1802, 			 Length:=1, Writable:=FALSE, Default_Value:=6, 		SubElements:=E_SubElement_types.With_fix_subelements);
	TPDO3_communication_parameter_COB_ID_used_by_TPDO					: ST_CAN_Object := (Name:='TPDO communication parameter_COB-ID used by TPDO', 					Index:=16#1802, Subindex:=1, 													SubElements:=E_SubElement_types.Fix_subelement);
	TPDO3_communication_parameter_Transmission_type						: ST_CAN_Object := (Name:='TPDO communication parameter_Transmission type', 					Index:=16#1802, Subindex:=2, Length:=1, 										SubElements:=E_SubElement_types.Fix_subelement);
	TPDO3_communication_parameter_Inhibit_time							: ST_CAN_Object := (Name:='TPDO communication parameter_Inhibit time', 							Index:=16#1802, Subindex:=3, Length:=2, 										SubElements:=E_SubElement_types.Fix_subelement);
	TPDO3_communication_parameter_Event_timer							: ST_CAN_Object := (Name:='TPDO communication parameter_Event timer', 							Index:=16#1802, Subindex:=5, Length:=2, 										SubElements:=E_SubElement_types.Fix_subelement);
	TPDO3_communication_parameter_SYNC_start_value						: ST_CAN_Object := (Name:='TPDO communication parameter_SYNC start value', 						Index:=16#1802, Subindex:=6, Length:=1, 										SubElements:=E_SubElement_types.Fix_subelement);
	TPDO4_communication_parameter_Highest_sub_index_supported			: ST_CAN_Object := (Name:='TPDO communication parameter_Highest sub-index supported', 			Index:=16#1803, 			 Length:=1, Writable:=FALSE, Default_Value:=6, 		SubElements:=E_SubElement_types.With_fix_subelements);
	TPDO4_communication_parameter_COB_ID_used_by_TPDO					: ST_CAN_Object := (Name:='TPDO communication parameter_COB-ID used by TPDO', 					Index:=16#1803, Subindex:=1, 													SubElements:=E_SubElement_types.Fix_subelement);
	TPDO4_communication_parameter_Transmission_type						: ST_CAN_Object := (Name:='TPDO communication parameter_Transmission type', 					Index:=16#1803, Subindex:=2, Length:=1, 										SubElements:=E_SubElement_types.Fix_subelement);
	TPDO4_communication_parameter_Inhibit_time							: ST_CAN_Object := (Name:='TPDO communication parameter_Inhibit time', 							Index:=16#1803, Subindex:=3, Length:=2, 										SubElements:=E_SubElement_types.Fix_subelement);
	TPDO4_communication_parameter_Event_timer							: ST_CAN_Object := (Name:='TPDO communication parameter_Event timer', 							Index:=16#1803, Subindex:=5, Length:=2, 										SubElements:=E_SubElement_types.Fix_subelement);
	TPDO4_communication_parameter_SYNC_start_value						: ST_CAN_Object := (Name:='TPDO communication parameter_SYNC start value', 						Index:=16#1803, Subindex:=6, Length:=1, 										SubElements:=E_SubElement_types.Fix_subelement);
	TPDO1_mapping_parameter_Number_of_mapped_application_objects_in_PDO	: ST_CAN_Object := (Name:='TPDO mapping parameter_Number of mapped application objects in PDO', Index:=16#1A00, 			 Length:=1, 										SubElements:=E_SubElement_types.With_fix_subelements);
	TPDO1_mapping_parameter_Application_object_1						: ST_CAN_Object := (Name:='TPDO mapping parameter_Application object 1', 						Index:=16#1A00, Subindex:=1, 													SubElements:=E_SubElement_types.Fix_subelement);
	TPDO1_mapping_parameter_Application_object_2						: ST_CAN_Object := (Name:='TPDO mapping parameter_Application object 2', 						Index:=16#1A00, Subindex:=2, 													SubElements:=E_SubElement_types.Fix_subelement);
	TPDO1_mapping_parameter_Application_object_3						: ST_CAN_Object := (Name:='TPDO mapping parameter_Application object 3', 						Index:=16#1A00, Subindex:=3, 													SubElements:=E_SubElement_types.Fix_subelement);
	TPDO1_mapping_parameter_Application_object_4						: ST_CAN_Object := (Name:='TPDO mapping parameter_Application object 4', 						Index:=16#1A00, Subindex:=4, 													SubElements:=E_SubElement_types.Fix_subelement);
	TPDO1_mapping_parameter_Application_object_5						: ST_CAN_Object := (Name:='TPDO mapping parameter_Application object 5',				 		Index:=16#1A00, Subindex:=5, 													SubElements:=E_SubElement_types.Fix_subelement);
	TPDO1_mapping_parameter_Application_object_6						: ST_CAN_Object := (Name:='TPDO mapping parameter_Application object 6', 						Index:=16#1A00, Subindex:=6, 													SubElements:=E_SubElement_types.Fix_subelement);
	TPDO1_mapping_parameter_Application_object_7						: ST_CAN_Object := (Name:='TPDO mapping parameter_Application object 7', 						Index:=16#1A00, Subindex:=7, 													SubElements:=E_SubElement_types.Fix_subelement);
	TPDO1_mapping_parameter_Application_object_8						: ST_CAN_Object := (Name:='TPDO mapping parameter_Application object 8',						Index:=16#1A00, Subindex:=8, 													SubElements:=E_SubElement_types.Fix_subelement);
	TPDO2_mapping_parameter_Number_of_mapped_application_objects_in_PDO	: ST_CAN_Object := (Name:='TPDO mapping parameter_Number of mapped application objects in PDO', Index:=16#1A01, 			 Length:=1,											SubElements:=E_SubElement_types.With_fix_subelements);
	TPDO2_mapping_parameter_Application_object_1						: ST_CAN_Object := (Name:='TPDO mapping parameter_Application object 1', 						Index:=16#1A01, Subindex:=1, 													SubElements:=E_SubElement_types.Fix_subelement);
	TPDO2_mapping_parameter_Application_object_2						: ST_CAN_Object := (Name:='TPDO mapping parameter_Application object 2', 						Index:=16#1A01, Subindex:=2, 													SubElements:=E_SubElement_types.Fix_subelement);
	TPDO2_mapping_parameter_Application_object_3						: ST_CAN_Object := (Name:='TPDO mapping parameter_Application object 3', 						Index:=16#1A01, Subindex:=3, 													SubElements:=E_SubElement_types.Fix_subelement);
	TPDO2_mapping_parameter_Application_object_4						: ST_CAN_Object := (Name:='TPDO mapping parameter_Application object 4', 						Index:=16#1A01, Subindex:=4, 													SubElements:=E_SubElement_types.Fix_subelement);
	TPDO2_mapping_parameter_Application_object_5						: ST_CAN_Object := (Name:='TPDO mapping parameter_Application object 5', 						Index:=16#1A01, Subindex:=5, 													SubElements:=E_SubElement_types.Fix_subelement);
	TPDO2_mapping_parameter_Application_object_6						: ST_CAN_Object := (Name:='TPDO mapping parameter_Application object 6', 						Index:=16#1A01, Subindex:=6, 													SubElements:=E_SubElement_types.Fix_subelement);
	TPDO2_mapping_parameter_Application_object_7						: ST_CAN_Object := (Name:='TPDO mapping parameter_Application object 7', 						Index:=16#1A01, Subindex:=7, 													SubElements:=E_SubElement_types.Fix_subelement);
	TPDO2_mapping_parameter_Application_object_8						: ST_CAN_Object := (Name:='TPDO mapping parameter_Application object 8', 						Index:=16#1A01, Subindex:=8, 													SubElements:=E_SubElement_types.Fix_subelement);
	TPDO3_mapping_parameter_Number_of_mapped_application_objects_in_PDO	: ST_CAN_Object := (Name:='TPDO mapping parameter_Number of mapped application objects in PDO', Index:=16#1A02, 			 Length:=1, 										SubElements:=E_SubElement_types.With_fix_subelements);
	TPDO3_mapping_parameter_Application_object_1						: ST_CAN_Object := (Name:='TPDO mapping parameter_Application object 1', 						Index:=16#1A02, Subindex:=1, 													SubElements:=E_SubElement_types.Fix_subelement);
	TPDO3_mapping_parameter_Application_object_2						: ST_CAN_Object := (Name:='TPDO mapping parameter_Application object 2', 						Index:=16#1A02, Subindex:=2, 													SubElements:=E_SubElement_types.Fix_subelement);
	TPDO3_mapping_parameter_Application_object_3						: ST_CAN_Object := (Name:='TPDO mapping parameter_Application object 3', 						Index:=16#1A02, Subindex:=3, 													SubElements:=E_SubElement_types.Fix_subelement);
	TPDO3_mapping_parameter_Application_object_4						: ST_CAN_Object := (Name:='TPDO mapping parameter_Application object 4', 						Index:=16#1A02, Subindex:=4, 													SubElements:=E_SubElement_types.Fix_subelement);
	TPDO3_mapping_parameter_Application_object_5						: ST_CAN_Object := (Name:='TPDO mapping parameter_Application object 5', 						Index:=16#1A02, Subindex:=5, 													SubElements:=E_SubElement_types.Fix_subelement);
	TPDO3_mapping_parameter_Application_object_6						: ST_CAN_Object := (Name:='TPDO mapping parameter_Application object 6', 						Index:=16#1A02, Subindex:=6, 													SubElements:=E_SubElement_types.Fix_subelement);
	TPDO3_mapping_parameter_Application_object_7						: ST_CAN_Object := (Name:='TPDO mapping parameter_Application object 7', 						Index:=16#1A02, Subindex:=7, 													SubElements:=E_SubElement_types.Fix_subelement);
	TPDO3_mapping_parameter_Application_object_8						: ST_CAN_Object := (Name:='TPDO mapping parameter_Application object 8', 						Index:=16#1A02, Subindex:=8, 													SubElements:=E_SubElement_types.Fix_subelement);
	TPDO4_mapping_parameter_Number_of_mapped_application_objects_in_PDO	: ST_CAN_Object := (Name:='TPDO mapping parameter_Number of mapped application objects in PDO', Index:=16#1A03, 			 Length:=1, 										SubElements:=E_SubElement_types.With_fix_subelements);
	TPDO4_mapping_parameter_Application_object_1						: ST_CAN_Object := (Name:='TPDO mapping parameter_Application object 1', 						Index:=16#1A03, Subindex:=1, 													SubElements:=E_SubElement_types.Fix_subelement);
	TPDO4_mapping_parameter_Application_object_2						: ST_CAN_Object := (Name:='TPDO mapping parameter_Application object 2', 						Index:=16#1A03, Subindex:=2, 													SubElements:=E_SubElement_types.Fix_subelement);
	TPDO4_mapping_parameter_Application_object_3						: ST_CAN_Object := (Name:='TPDO mapping parameter_Application object 3', 						Index:=16#1A03, Subindex:=3, 													SubElements:=E_SubElement_types.Fix_subelement);
	TPDO4_mapping_parameter_Application_object_4						: ST_CAN_Object := (Name:='TPDO mapping parameter_Application object 4', 						Index:=16#1A03, Subindex:=4, 													SubElements:=E_SubElement_types.Fix_subelement);
	TPDO4_mapping_parameter_Application_object_5						: ST_CAN_Object := (Name:='TPDO mapping parameter_Application object 5', 						Index:=16#1A03, Subindex:=5, 													SubElements:=E_SubElement_types.Fix_subelement);
	TPDO4_mapping_parameter_Application_object_6						: ST_CAN_Object := (Name:='TPDO mapping parameter_Application object 6', 						Index:=16#1A03, Subindex:=6, 													SubElements:=E_SubElement_types.Fix_subelement);
	TPDO4_mapping_parameter_Application_object_7						: ST_CAN_Object := (Name:='TPDO mapping parameter_Application object 7', 						Index:=16#1A03, Subindex:=7, 													SubElements:=E_SubElement_types.Fix_subelement);
	TPDO4_mapping_parameter_Application_object_8						: ST_CAN_Object := (Name:='TPDO mapping parameter_Application object 8', 						Index:=16#1A03, Subindex:=8, 													SubElements:=E_SubElement_types.Fix_subelement);
END_VAR

// ---- GVLs/DS302_Object_List.TcGVL
{attribute 'qualified_only'}
VAR_GLOBAL
	Download_Program_Data_Number_of_entries							: ST_CAN_Object := (Name:='Download Program Data_Number of entries', 							Index:=16#1F50, 			 Length:=1, 	Writable:=FALSE,	Default_Value:=1);
	Download_Program_Data_Program_Area								: ST_CAN_Object := (Name:='Download Program Data_Program Area', 								Index:=16#1F50, Subindex:=1, Length:=255);
	Program_Control_Number_of_entries								: ST_CAN_Object := (Name:='Program Control_Number of entries', 									Index:=16#1F51,				 Length:=1, 	Writable:=FALSE,	Default_Value:=1);
	Program_Control_Program_Control									: ST_CAN_Object := (Name:='Program Control_Program Control', 									Index:=16#1F51, Subindex:=1, Length:=1);
	Program_Software_Identification_Number_of_entries				: ST_CAN_Object := (Name:='Program Software Identification_Number of entries', 					Index:=16#1F56,				 Length:=1, 	Writable:=FALSE,	Default_Value:=1);
	Program_Software_Identification_Program_Software_Identification	: ST_CAN_Object := (Name:='Program Software Identification_Program Software Identification', 	Index:=16#1F56, Subindex:=1,			 	Writable:=FALSE);
	Flash_Status_Identification_Number_of_entries					: ST_CAN_Object := (Name:='Flash Status Identification_Number of entries', 						Index:=16#1F57,				 Length:=1, 	Writable:=FALSE,	Default_Value:=1);
	Flash_Status_Identification_Flash_Status						: ST_CAN_Object := (Name:='Flash Status Identification_Flash Status', 							Index:=16#1F57, Subindex:=1,			 	Writable:=FALSE);
	Firmware_Data_Identification_Number_of_entries					: ST_CAN_Object := (Name:='Firmware Data Identification_Number of entries', 					Index:=16#1F5A,				 Length:=1, 	Writable:=FALSE,	Default_Value:=3);
	Firmware_Data_Identification_Project_Id							: ST_CAN_Object := (Name:='Firmware Data Identification_Project Id', 							Index:=16#1F5A, Subindex:=1, Length:=255);
	Firmware_Data_Identification_Firmware_Id						: ST_CAN_Object := (Name:='Firmware Data Identification_Firmware Id', 							Index:=16#1F5A, Subindex:=2, Length:=1, 	Writable:=FALSE,	Default_Value:=1);
	Firmware_Data_Identification_Max_Block_Size						: ST_CAN_Object := (Name:='Firmware Data Identification_Max Block Size', 						Index:=16#1F5A, Subindex:=3, Length:=2, 	Writable:=FALSE,	Default_Value:=256);
END_VAR

// ---- GVLs/DS402_Object_List.TcGVL
{attribute 'qualified_only'}
VAR_GLOBAL
	Abort_connection_option_code									: ST_CAN_Object := (Name:='Abort connection option code', 							Index:=16#6007,				 Length:=2,												Default_Value:=1);
	Error_code														: ST_CAN_Object := (Name:='Error code', 											Index:=16#603F,				 Length:=2, Writable:=FALSE,	TPDO_Mappable:=TRUE);
	
	Controlword														: ST_CAN_Object	:= (Name:='Controlword', 											Index:=16#6040,				 Length:=2,						RPDO_Mappable:=TRUE);
	Statusword														: ST_CAN_Object := (Name:='Statusword', 											Index:=16#6041,				 Length:=2, Writable:=FALSE,	TPDO_Mappable:=TRUE);
	vl_target_velocity												: ST_CAN_Object	:= (Name:='vl target velocity', 									Index:=16#6042,				 Length:=2,						RPDO_Mappable:=TRUE);
	vl_velocity_demand												: ST_CAN_Object	:= (Name:='vl velocity demand', 									Index:=16#6043,				 Length:=2, Writable:=FALSE,	TPDO_Mappable:=TRUE);
	vl_velocity_actual_value										: ST_CAN_Object := (Name:='vl velocity actual value', 								Index:=16#6044,				 Length:=2, Writable:=FALSE,	TPDO_Mappable:=TRUE);
	vl_velocity_min_max_amount_Highest_sub_index_supported			: ST_CAN_Object := (Name:='vl velocity min max amount_Highest sub-index supported',	Index:=16#6046,				 Length:=1, Writable:=FALSE, 							Default_Value:=2,	SubElements:=E_SubElement_types.With_fix_subelements);
	vl_velocity_min_max_amount_vl_velocity_min_amount				: ST_CAN_Object := (Name:='vl velocity min max amount_vl velocity min amount', 		Index:=16#6046, Subindex:=1, 								RPDO_Mappable:=TRUE, 						SubElements:=E_SubElement_types.Fix_subelement);
	vl_velocity_min_max_amount_vl_velocity_max_amount				: ST_CAN_Object := (Name:='vl velocity min max amount_vl velocity max amount', 		Index:=16#6046, Subindex:=2, 								RPDO_Mappable:=TRUE, 						SubElements:=E_SubElement_types.Fix_subelement);
	vl_velocity_acceleration_Highest_sub_index_supported			: ST_CAN_Object := (Name:='vl velocity acceleration_Highest sub-index supported', 	Index:=16#6048,				 Length:=1, Writable:=FALSE, 							Default_Value:=2,	SubElements:=E_SubElement_types.With_fix_subelements);
	vl_velocity_acceleration_Delta_speed							: ST_CAN_Object := (Name:='vl velocity acceleration_Delta speed', 					Index:=16#6048, Subindex:=1, 								RPDO_Mappable:=TRUE, 						SubElements:=E_SubElement_types.Fix_subelement);
	vl_velocity_acceleration_Delta_time								: ST_CAN_Object := (Name:='vl velocity acceleration_Delta time', 					Index:=16#6048, Subindex:=2, Length:=2, 					RPDO_Mappable:=TRUE, 						SubElements:=E_SubElement_types.Fix_subelement);
	vl_velocity_deceleration_Highest_sub_index_supported			: ST_CAN_Object := (Name:='vl velocity deceleration_Highest sub-index supported', 	Index:=16#6049,				 Length:=1, Writable:=FALSE, 							Default_Value:=2,	SubElements:=E_SubElement_types.With_fix_subelements);
	vl_velocity_deceleration_Delta_speed							: ST_CAN_Object := (Name:='vl velocity deceleration_Delta speed', 					Index:=16#6049, Subindex:=1, 								RPDO_Mappable:=TRUE, 						SubElements:=E_SubElement_types.Fix_subelement);
	vl_velocity_deceleration_Delta_time								: ST_CAN_Object := (Name:='vl velocity deceleration_Delta time', 					Index:=16#6049, Subindex:=2, Length:=2, 					RPDO_Mappable:=TRUE, 						SubElements:=E_SubElement_types.Fix_subelement);
	vl_velocity_quick_stop_Highest_sub_index_supported				: ST_CAN_Object := (Name:='vl velocity quick stop_Highest sub-index supported', 	Index:=16#604A,				 Length:=1, Writable:=FALSE, 							Default_Value:=2,	SubElements:=E_SubElement_types.With_fix_subelements);
	vl_velocity_quick_stop_Delta_speed								: ST_CAN_Object := (Name:='vl velocity quick stop_Delta speed', 					Index:=16#604A, Subindex:=1, 								RPDO_Mappable:=TRUE, 						SubElements:=E_SubElement_types.Fix_subelement);
	vl_velocity_quick_stop_Delta_time								: ST_CAN_Object := (Name:='vl velocity quick stop_Delta time', 						Index:=16#604A, Subindex:=2, Length:=2, 					RPDO_Mappable:=TRUE, 						SubElements:=E_SubElement_types.Fix_subelement);
	vl_set_point_factor_Highest_sub_index_supported					: ST_CAN_Object := (Name:='vl set-point factor_Highest sub-index supported', 		Index:=16#604B,				 Length:=1, Writable:=FALSE, 							Default_Value:=2,	SubElements:=E_SubElement_types.With_fix_subelements);
	vl_set_point_factor_Numerator									: ST_CAN_Object := (Name:='vl set-point factor_Numerator', 							Index:=16#604B, Subindex:=1, 								RPDO_Mappable:=TRUE, 						SubElements:=E_SubElement_types.Fix_subelement);
	vl_set_point_factor_Denominator									: ST_CAN_Object := (Name:='vl set-point factor_Denominator', 						Index:=16#604B, Subindex:=2, Length:=2, 					RPDO_Mappable:=TRUE, 						SubElements:=E_SubElement_types.Fix_subelement);
	vl_dimension_factor_Highest_sub_index_supported					: ST_CAN_Object := (Name:='vl dimension factor_Highest sub-index supported', 		Index:=16#604C,				 Length:=1,	Writable:=FALSE, 							Default_Value:=2,	SubElements:=E_SubElement_types.With_fix_subelements);
	vl_dimension_factor_Numerator									: ST_CAN_Object := (Name:='vl dimension factor_Numerator', 							Index:=16#604C, Subindex:=1, 								RPDO_Mappable:=TRUE, 						SubElements:=E_SubElement_types.Fix_subelement);
	vl_dimension_factor_Denominator									: ST_CAN_Object := (Name:='vl dimension factor_Denominator', 						Index:=16#604C, Subindex:=2, Length:=2, 					RPDO_Mappable:=TRUE, 						SubElements:=E_SubElement_types.Fix_subelement);
	
	Quick_stop_option_code											: ST_CAN_Object := (Name:='Quick stop option code', 								Index:=16#605A,				 Length:=2,												Default_Value:=2);
	Shutdown_option_code											: ST_CAN_Object := (Name:='Shutdown option code', 									Index:=16#605B,				 Length:=2);
	Disable_operation_option_code									: ST_CAN_Object := (Name:='Disable operation option code', 							Index:=16#605C,				 Length:=2,												Default_Value:=1);
	Halt_option_code												: ST_CAN_Object := (Name:='Halt option code', 										Index:=16#605D,				 Length:=2,												Default_Value:=1);
	Fault_reaction_option_code										: ST_CAN_Object := (Name:='Fault reaction option code', 							Index:=16#605E,				 Length:=2,												Default_Value:=2);

	Modes_of_operation												: ST_CAN_Object := (Name:='Modes of operation', 									Index:=16#6060,				 Length:=1,						RPDO_Mappable:=TRUE);
	Modes_of_operation_display										: ST_CAN_Object := (Name:='Modes of operation display', 							Index:=16#6061,				 Length:=1, Writable:=FALSE,	TPDO_Mappable:=TRUE);
	Position_demand_value											: ST_CAN_Object := (Name:='Position demand value', 									Index:=16#6062,				 			Writable:=FALSE,	TPDO_Mappable:=TRUE);
	Position_actual_internal_value									: ST_CAN_Object := (Name:='Position actual internal value', 						Index:=16#6063,				 			Writable:=FALSE,	TPDO_Mappable:=TRUE);
	Position_actual_value											: ST_CAN_Object := (Name:='Position actual value', 									Index:=16#6064,				 			Writable:=FALSE,	TPDO_Mappable:=TRUE);
	Following_error_window											: ST_CAN_Object := (Name:='Following error window', 								Index:=16#6065,				 								RPDO_Mappable:=TRUE);
	Following_error_time_out										: ST_CAN_Object := (Name:='Following error time out', 								Index:=16#6066,				 Length:=2,						RPDO_Mappable:=TRUE);
	Position_window													: ST_CAN_Object := (Name:='Position window', 										Index:=16#6067,				 								RPDO_Mappable:=TRUE);
	Position_window_time											: ST_CAN_Object := (Name:='Position window time', 									Index:=16#6068,				 Length:=2,						RPDO_Mappable:=TRUE);
	Velocity_sensor_actual_value									: ST_CAN_Object := (Name:='Velocity sensor actual value', 							Index:=16#6069,				 			Writable:=FALSE,	TPDO_Mappable:=TRUE);
	Sensor_selection_code											: ST_CAN_Object := (Name:='Sensor selection code', 									Index:=16#606A,				 			Writable:=FALSE,	RPDO_Mappable:=TRUE);
	Velocity_demand_value											: ST_CAN_Object := (Name:='Velocity demand value', 									Index:=16#606B,				 			Writable:=FALSE,	TPDO_Mappable:=TRUE);
	Velocity_actual_value											: ST_CAN_Object := (Name:='Velocity actual value', 									Index:=16#606C,				 			Writable:=FALSE,	TPDO_Mappable:=TRUE);
	Velocity_window													: ST_CAN_Object := (Name:='Velocity window', 										Index:=16#606D,				 Length:=2,						RPDO_Mappable:=TRUE);
	Velocity_window_time											: ST_CAN_Object := (Name:='Velocity window time', 									Index:=16#606E,				 Length:=2,						RPDO_Mappable:=TRUE);
	Velocity_threshold												: ST_CAN_Object := (Name:='Velocity threshold', 									Index:=16#606F,				 Length:=2,						RPDO_Mappable:=TRUE);
	
	Velocity_threshold_time											: ST_CAN_Object := (Name:='Velocity threshold time', 								Index:=16#6070,				 Length:=2,						RPDO_Mappable:=TRUE);
	Target_torque													: ST_CAN_Object := (Name:='Target torque', 											Index:=16#6071,				 Length:=2,						RPDO_Mappable:=TRUE);
	Max_torque														: ST_CAN_Object := (Name:='Max torque', 											Index:=16#6072,				 Length:=2,						RPDO_Mappable:=TRUE);
	Max_current														: ST_CAN_Object := (Name:='Max current', 											Index:=16#6073,				 Length:=2,						RPDO_Mappable:=TRUE);
	Torque_demand													: ST_CAN_Object := (Name:='Torque demand', 											Index:=16#6074,				 Length:=2,	Writable:=FALSE,	TPDO_Mappable:=TRUE);
	Motor_rated_current												: ST_CAN_Object := (Name:='Motor rated current', 									Index:=16#6075);
	Motor_rated_torque												: ST_CAN_Object := (Name:='Motor rated torque', 									Index:=16#6076);
	Torque_actual_value												: ST_CAN_Object := (Name:='Torque actual value',	 								Index:=16#6077,				 Length:=2,	Writable:=FALSE,	TPDO_Mappable:=TRUE);
	Current_actual_value											: ST_CAN_Object := (Name:='Current actual value', 									Index:=16#6078,				 Length:=2,	Writable:=FALSE,	TPDO_Mappable:=TRUE);
	DC_link_circuit_voltage											: ST_CAN_Object := (Name:='DC link circuit voltage', 								Index:=16#6079,				 			Writable:=FALSE,	TPDO_Mappable:=TRUE);
	Target_position													: ST_CAN_Object := (Name:='Target position', 										Index:=16#607A,				 								RPDO_Mappable:=TRUE);
	Position_range_limit_Highest_sub_index_supported				: ST_CAN_Object := (Name:='Position range limit_Highest sub-index supported', 		Index:=16#607B,				 Length:=1, Writable:=FALSE,							Default_Value:=2, 	SubElements:=E_SubElement_types.With_fix_subelements);
	Position_range_limit_Min_position_range_limit					: ST_CAN_Object := (Name:='Position range limit_Min position range limit',			Index:=16#607B, Subindex:=1, 								RPDO_Mappable:=TRUE,						SubElements:=E_SubElement_types.Fix_subelement);
	Position_range_limit_Max_position_range_limit					: ST_CAN_Object := (Name:='Position range limit_Max position range limit',			Index:=16#607B, Subindex:=2, 								RPDO_Mappable:=TRUE, 						SubElements:=E_SubElement_types.Fix_subelement);
	Home_offset														: ST_CAN_Object := (Name:='Home offset', 											Index:=16#607C,				 								RPDO_Mappable:=TRUE);
	Software_position_limit_Highest_sub_index_supported				: ST_CAN_Object := (Name:='Software position limit_Highest sub-index supported', 	Index:=16#607D,				 Length:=1, Writable:=FALSE,							Default_Value:=2, 	SubElements:=E_SubElement_types.With_fix_subelements);
	Software_position_limit_Min_position_limit						: ST_CAN_Object := (Name:='Software position limit_Min position limit',		 		Index:=16#607D, Subindex:=1, 								RPDO_Mappable:=TRUE, 						SubElements:=E_SubElement_types.Fix_subelement);
	Software_position_limit_Max_position_limit						: ST_CAN_Object := (Name:='Software position limit_Max position limit', 			Index:=16#607D, Subindex:=2, 								RPDO_Mappable:=TRUE, 						SubElements:=E_SubElement_types.Fix_subelement);
	Polarity														: ST_CAN_Object := (Name:='Polarity', 												Index:=16#607E,				 Length:=1,						RPDO_Mappable:=TRUE);
	Max_profile_velocity											: ST_CAN_Object := (Name:='Max profile velocity', 									Index:=16#607F,				 								RPDO_Mappable:=TRUE);
	
	Max_motor_speed													: ST_CAN_Object := (Name:='Max motor speed',	 									Index:=16#6080,				 								RPDO_Mappable:=TRUE);
	Profile_velocity												: ST_CAN_Object := (Name:='Profile velocity', 										Index:=16#6081,				 								RPDO_Mappable:=TRUE);
	End_velocity													: ST_CAN_Object := (Name:='End velocity', 											Index:=16#6082,				 								RPDO_Mappable:=TRUE);
	Profile_acceleration											: ST_CAN_Object := (Name:='Profile acceleration', 									Index:=16#6083,				 								RPDO_Mappable:=TRUE);
	Profile_deceleration											: ST_CAN_Object := (Name:='Profile deceleration', 									Index:=16#6084,				 								RPDO_Mappable:=TRUE);
	Quick_stop_deceleration											: ST_CAN_Object := (Name:='Quick stop deceleration', 								Index:=16#6085,				 								RPDO_Mappable:=TRUE);
	Motion_profile_type												: ST_CAN_Object := (Name:='Motion profile type', 									Index:=16#6086,				 Length:=2,						RPDO_Mappable:=TRUE);
	Torque_slope													: ST_CAN_Object := (Name:='Torque slope', 											Index:=16#6087,				 								RPDO_Mappable:=TRUE);
	Torque_profile_type												: ST_CAN_Object := (Name:='Torque profile type', 									Index:=16#6088,				 Length:=2,				 		RPDO_Mappable:=TRUE);
	Position_encoder_resolution_Highest_sub_index_supported			: ST_CAN_Object := (Name:='Position encoder resolution_Highest sub-index supported',Index:=16#608F,				 Length:=1, Writable:=FALSE, 							Default_Value:=2, 	SubElements:=E_SubElement_types.With_fix_subelements);
	Position_encoder_resolution_Encoder_increments					: ST_CAN_Object := (Name:='Position encoder resolution_Encoder increments', 		Index:=16#608F, Subindex:=1, 						 		RPDO_Mappable:=TRUE,						SubElements:=E_SubElement_types.Fix_subelement);
	Position_encoder_resolution_Motor_revolutions					: ST_CAN_Object := (Name:='Position encoder resolution_Motor revolutions', 			Index:=16#608F, Subindex:=2, 						 		RPDO_Mappable:=TRUE,						SubElements:=E_SubElement_types.Fix_subelement);
	
	Velocity_encoder_resolution_Highest_sub_index_supported			: ST_CAN_Object := (Name:='Velocity encoder resolution_Highest sub-index supported',Index:=16#6090,				 Length:=1, Writable:=FALSE, 							Default_Value:=2, 	SubElements:=E_SubElement_types.With_fix_subelements);
	Velocity_encoder_resolution_Encoder_increments					: ST_CAN_Object := (Name:='Velocity encoder resolution_Encoder increments', 		Index:=16#6090, Subindex:=1, 						 		RPDO_Mappable:=TRUE, 						SubElements:=E_SubElement_types.Fix_subelement);
	Velocity_encoder_resolution_Motor_revolutions					: ST_CAN_Object := (Name:='Velocity encoder resolution_Motor revolutions', 			Index:=16#6090, Subindex:=2, 						 		RPDO_Mappable:=TRUE, 						SubElements:=E_SubElement_types.Fix_subelement);
	Gear_ratio_Highest_sub_index_supported							: ST_CAN_Object := (Name:='Gear ratio_Highest sub-index supported', 				Index:=16#6091,				 Length:=1, Writable:=FALSE, 							Default_Value:=2, 	SubElements:=E_SubElement_types.With_fix_subelements);
	Gear_ratio_Motor_shaft_revolutions								: ST_CAN_Object := (Name:='Gear ratio_Motor shaft revolutions', 					Index:=16#6091, Subindex:=1, 						 		RPDO_Mappable:=TRUE, 						SubElements:=E_SubElement_types.Fix_subelement);
	Gear_ratio_Driving_shaft_revolutions							: ST_CAN_Object := (Name:='Gear ratio_Driving shaft revolutions',				 	Index:=16#6091, Subindex:=2, 						 		RPDO_Mappable:=TRUE, 						SubElements:=E_SubElement_types.Fix_subelement);
	Feed_constant_Highest_sub_index_supported						: ST_CAN_Object := (Name:='Feed constant_Highest sub-index supported', 				Index:=16#6092,				 Length:=1, Writable:=FALSE, 							Default_Value:=2, 	SubElements:=E_SubElement_types.With_fix_subelements);
	Feed_constant_Feed												: ST_CAN_Object := (Name:='Feed constant_Feed', 									Index:=16#6092, Subindex:=1, 						 		RPDO_Mappable:=TRUE, 						SubElements:=E_SubElement_types.Fix_subelement);
	Feed_constant_Shaft_Revolution									: ST_CAN_Object := (Name:='Feed constant_Shaft Revolution', 						Index:=16#6092, Subindex:=2, 						 		RPDO_Mappable:=TRUE, 						SubElements:=E_SubElement_types.Fix_subelement);
	Velocity_Factor_Highest_sub_index_supported						: ST_CAN_Object := (Name:='Velocity Factor_Highest sub-index supported', 			Index:=16#6096,				 Length:=1, Writable:=FALSE, 							Default_Value:=2, 	SubElements:=E_SubElement_types.With_fix_subelements);
	Velocity_Factor_Numerator										: ST_CAN_Object := (Name:='Velocity Factor_Numerator', 								Index:=16#6096, Subindex:=1, 						 		RPDO_Mappable:=TRUE, 	Default_Value:=1, 	SubElements:=E_SubElement_types.Fix_subelement);
	Velocity_Factor_Divisor											: ST_CAN_Object := (Name:='Velocity Factor_Divisor', 								Index:=16#6096, Subindex:=2, 						 		RPDO_Mappable:=TRUE, 	Default_Value:=1, 	SubElements:=E_SubElement_types.Fix_subelement);
	Acceleration_Factor_Highest_sub_index_supported					: ST_CAN_Object := (Name:='Acceleration Factor_Highest sub-index supported', 		Index:=16#6097,				 Length:=1, Writable:=FALSE, 							Default_Value:=2, 	SubElements:=E_SubElement_types.With_fix_subelements);
	Acceleration_Factor_Numerator									: ST_CAN_Object := (Name:='Acceleration Factor_Numerator', 							Index:=16#6097, Subindex:=1, 						 		RPDO_Mappable:=TRUE, 	Default_Value:=1, 	SubElements:=E_SubElement_types.Fix_subelement);
	Acceleration_Factor_Divisor										: ST_CAN_Object := (Name:='Acceleration Factor_Divisor', 							Index:=16#6097, Subindex:=2, 						 		RPDO_Mappable:=TRUE, 	Default_Value:=1, 	SubElements:=E_SubElement_types.Fix_subelement);
	Homing_method													: ST_CAN_Object := (Name:='Homing method', 											Index:=16#6098,				 Length:=1,				 		RPDO_Mappable:=TRUE);
	Homing_speeds_Highest_sub_index_supported						: ST_CAN_Object := (Name:='Homing speeds_Highest sub-index supported', 				Index:=16#6099,				 Length:=1, Writable:=FALSE,							Default_Value:=2, 	SubElements:=E_SubElement_types.With_fix_subelements);
	Homing_speeds_Speed_during_search_for_switch					: ST_CAN_Object := (Name:='Homing speeds_Speed during search for switch',			Index:=16#6099, Subindex:=1, 						 		RPDO_Mappable:=TRUE, 						SubElements:=E_SubElement_types.Fix_subelement);
	Homing_speeds_Speed_during_search_for_zero						: ST_CAN_Object := (Name:='Homing speeds_Speed during search for zero', 			Index:=16#6099, Subindex:=2, 						 		RPDO_Mappable:=TRUE, 						SubElements:=E_SubElement_types.Fix_subelement);
	Homing_acceleration												: ST_CAN_Object := (Name:='Homing acceleration', 									Index:=16#609A,				 								RPDO_Mappable:=TRUE);
	
	Jerk_factor_Factor_Highest_sub_index_supported					: ST_CAN_Object := (Name:='Jerk factor Factor_Highest sub-index supported', 		Index:=16#60A2,				 Length:=1, Writable:=FALSE, 							Default_Value:=2,	SubElements:=E_SubElement_types.With_fix_subelements);
	Jerk_factor_Factor_Numerator									: ST_CAN_Object := (Name:='Jerk factor Factor_Numerator', 							Index:=16#60A2, Subindex:=1, 														Default_Value:=1,	SubElements:=E_SubElement_types.Fix_subelement);
	Jerk_factor_Factor_Divisor										: ST_CAN_Object := (Name:='Jerk factor Factor_Divisor', 							Index:=16#60A2, Subindex:=2, 														Default_Value:=1,	SubElements:=E_SubElement_types.Fix_subelement);
	Profile_jerk_use												: ST_CAN_Object := (Name:='Profile jerk use', 										Index:=16#60A3,				 Length:=1);	
	Profile_jerk_Highest_sub_index_supported						: ST_CAN_Object := (Name:='Profile jerk_Highest sub-index supported', 				Index:=16#60A4,				 Length:=1, Writable:=FALSE,							Default_Value:=2, 	SubElements:=E_SubElement_types.With_list);
	Profile_jerk_1													: ST_CAN_Object := (Name:='Profile jerk 1', 										Index:=16#60A4, Subindex:=1, 																			SubElements:=E_SubElement_types.List_element);
	SI_unit_postion													: ST_CAN_Object := (Name:='SI unit postion', 										Index:=16#60A8);
	SI_unit_velocity												: ST_CAN_Object := (Name:='SI unit velocity', 										Index:=16#60A9);
	SI_unit_acceleration											: ST_CAN_Object := (Name:='SI unit acceleration', 									Index:=16#60AA);
	SI_unit_jerk													: ST_CAN_Object := (Name:='SI unit jerk', 											Index:=16#60AB);
	
	Position_offset													: ST_CAN_Object := (Name:='Position offset', 										Index:=16#60B0,				 								RPDO_Mappable:=TRUE);
	Velocity_offset													: ST_CAN_Object := (Name:='Velocity offset', 										Index:=16#60B1,				 								RPDO_Mappable:=TRUE);
	Torque_offset													: ST_CAN_Object := (Name:='Torque offset', 											Index:=16#60B2,				 Length:=2,				 		RPDO_Mappable:=TRUE);
	Touch_probe_mode												: ST_CAN_Object := (Name:='Touch probe mode', 										Index:=16#60B8,				 Length:=2,				 		RPDO_Mappable:=TRUE);
	Touch_probe_status												: ST_CAN_Object := (Name:='Touch probe status', 									Index:=16#60B9,				 Length:=2, Writable:=FALSE,	TPDO_Mappable:=TRUE);
	Touch_probe_1_positive_edge										: ST_CAN_Object := (Name:='Touch probe 1 positive edge', 							Index:=16#60BA,				 			Writable:=FALSE,	TPDO_Mappable:=TRUE);
	Touch_probe_1_negative_edge										: ST_CAN_Object := (Name:='Touch probe 1 negative edge', 							Index:=16#60BB,				 			Writable:=FALSE,	TPDO_Mappable:=TRUE);
	Touch_probe_2_positive_edge										: ST_CAN_Object := (Name:='Touch probe 2 positive edge', 							Index:=16#60BC,				 			Writable:=FALSE,	TPDO_Mappable:=TRUE);
	Touch_probe_2_negative_edge										: ST_CAN_Object := (Name:='Touch probe 2 negative edge', 							Index:=16#60BD,				 			Writable:=FALSE,	TPDO_Mappable:=TRUE);
	
	Interpolation_sub_mode_select									: ST_CAN_Object := (Name:='Interpolation sub mode select', 							Index:=16#60C0,				 Length:=2,				 		RPDO_Mappable:=TRUE);
	Interpolation_data_record_Highest_sub_index_supported			: ST_CAN_Object := (Name:='Interpolation data record_Highest sub-index supported',	Index:=16#60C1,				 Length:=1, Writable:=FALSE, 												SubElements:=E_SubElement_types.With_list);
	Interpolation_data_record_First_set_point						: ST_CAN_Object := (Name:='Interpolation data record_First set point', 				Index:=16#60C1, Subindex:=1, 								RPDO_Mappable:=TRUE, 						SubElements:=E_SubElement_types.List_element);
	Interpolation_time_period_Highest_sub_index_supported			: ST_CAN_Object := (Name:='Interpolation time period_Highest sub-index supported', 	Index:=16#60C2,				 Length:=1, Writable:=FALSE, 							Default_Value:=2, 	SubElements:=E_SubElement_types.With_fix_subelements);
	Interpolation_time_period_Interpolation_time_period_value		: ST_CAN_Object := (Name:='Interpolation time period_Interpolation time period value',Index:=16#60C2,Subindex:=1,Length:=1,				 		RPDO_Mappable:=TRUE,	Default_Value:=1, 	SubElements:=E_SubElement_types.Fix_subelement);
	Interpolation_time_period_Interpolation_time_index				: ST_CAN_Object := (Name:='Interpolation time period_Interpolation time index', 	Index:=16#60C2, Subindex:=2, Length:=1,				 		RPDO_Mappable:=TRUE,	Default_Value:=-3,	SubElements:=E_SubElement_types.Fix_subelement);
	Interpolation_data_configuration_Highest_sub_index_supported	: ST_CAN_Object := (Name:='Interpolation data configuration_Highest sub-index supported', Index:=16#60C4,		 Length:=1, Writable:=FALSE,							Default_Value:=6, 	SubElements:=E_SubElement_types.With_fix_subelements);
	Interpolation_data_configuration_Maximum_buffer_size 			: ST_CAN_Object := (Name:='Interpolation data configuration_Maximum buffer size', 	Index:=16#60C4, Subindex:=1, Length:=1, Writable:=FALSE, 												SubElements:=E_SubElement_types.Fix_subelement);
	Interpolation_data_configuration_Actual_buffer_size				: ST_CAN_Object := (Name:='Interpolation data configuration_Actual buffer size', 	Index:=16#60C4, Subindex:=2, Length:=1, Writable:=FALSE,	RPDO_Mappable:=TRUE, 						SubElements:=E_SubElement_types.Fix_subelement);
	Interpolation_data_configuration_Buffer_organisation 			: ST_CAN_Object := (Name:='Interpolation data configuration_Buffer organisation', 	Index:=16#60C4, Subindex:=3, Length:=1, Writable:=FALSE,	RPDO_Mappable:=TRUE, 						SubElements:=E_SubElement_types.Fix_subelement);
	Interpolation_data_configuration_Buffer_position				: ST_CAN_Object := (Name:='Interpolation data configuration_Buffer position', 		Index:=16#60C4, Subindex:=4, Length:=1, Writable:=FALSE,	RPDO_Mappable:=TRUE, 						SubElements:=E_SubElement_types.Fix_subelement);
	Interpolation_data_configuration_Size_of_data_record 			: ST_CAN_Object := (Name:='Interpolation data configuration_Size of data record', 	Index:=16#60C4, Subindex:=5, Length:=1, Writable:=FALSE,	RPDO_Mappable:=TRUE, 	Default_Value:=1, 	SubElements:=E_SubElement_types.Fix_subelement);
	Interpolation_data_configuration_Buffer_clear					: ST_CAN_Object := (Name:='Interpolation data configuration_Buffer clear', 			Index:=16#60C4, Subindex:=6, Length:=1, Writable:=FALSE,	RPDO_Mappable:=TRUE, 						SubElements:=E_SubElement_types.Fix_subelement);
	Max_acceleration												: ST_CAN_Object := (Name:='Max acceleration', 										Index:=16#60C5,				 								RPDO_Mappable:=TRUE);
	Max_deceleration												: ST_CAN_Object := (Name:='Max deceleration', 										Index:=16#60C6,				 								RPDO_Mappable:=TRUE);
		
	Touch_probe_source												: ST_CAN_Object := (Name:='Touch probe source',										Index:=16#60D0,				 Length:=2, Writable:=FALSE);
	Touch_probe_time_stamp_1_positive_value							: ST_CAN_Object := (Name:='Touch probe time stamp 1 positive value',	 			Index:=16#60D1,				 			Writable:=FALSE,	TPDO_Mappable:=TRUE);
	Touch_probe_time_stamp_1_negative_value							: ST_CAN_Object := (Name:='Touch probe time stamp 1 negative value', 				Index:=16#60D2,				 			Writable:=FALSE,	TPDO_Mappable:=TRUE);
	Touch_probe_time_stamp_2_positive_value							: ST_CAN_Object := (Name:='Touch probe time stamp 2 positive value', 				Index:=16#60D3,				 			Writable:=FALSE,	TPDO_Mappable:=TRUE);
	Touch_probe_time_stamp_2_negative_value							: ST_CAN_Object := (Name:='Touch probe time stamp 2 negative value', 				Index:=16#60D4,				 			Writable:=FALSE,	TPDO_Mappable:=TRUE);
	Touch_probe_1_positive_counter									: ST_CAN_Object := (Name:='Touch probe 1 positive counter', 						Index:=16#60D5,				 			Writable:=FALSE,	TPDO_Mappable:=TRUE);
	Touch_probe_1_negative_counter									: ST_CAN_Object := (Name:='Touch probe 1 negative counter', 						Index:=16#60D6,				 			Writable:=FALSE,	TPDO_Mappable:=TRUE);
	Touch_probe_2_positive_counter									: ST_CAN_Object := (Name:='Touch probe 2 positive counter', 						Index:=16#60D7,				 			Writable:=FALSE,	TPDO_Mappable:=TRUE);
	Touch_probe_2_negative_counter									: ST_CAN_Object := (Name:='Touch probe 2 negative counter', 						Index:=16#60D8,				 			Writable:=FALSE,	TPDO_Mappable:=TRUE);
	
	Positive_torque_limit_value										: ST_CAN_Object := (Name:='Positive torque limit value', 							Index:=16#60E0,				 Length:=2,						RPDO_Mappable:=TRUE);
	Negative_torque_limit_value										: ST_CAN_Object := (Name:='Negative torque limit value', 							Index:=16#60E1,				 Length:=2,						RPDO_Mappable:=TRUE);
	Supported_Homing_Methods_Highest_sub_index_supported			: ST_CAN_Object := (Name:='Supported Homing Methods_Highest sub-index supported', 	Index:=16#60E3,				 Length:=1, Writable:=FALSE,							Default_Value:=5, 	SubElements:=E_SubElement_types.With_list);
	Supported_Homing_Methods_Supported_homing_method_1				: ST_CAN_Object := (Name:='Supported Homing Methods_Supported homing method 1', 	Index:=16#60E3, Subindex:=1, Length:=1, Writable:=FALSE,							Default_Value:=37,	SubElements:=E_SubElement_types.List_element);
			
	Position_option_code											: ST_CAN_Object := (Name:='Position option code', 									Index:=16#60F2,				 Length:=2,						RPDO_Mappable:=TRUE);
	Following_error_actual_value									: ST_CAN_Object := (Name:='Following error actual value', 							Index:=16#60F4,				 			Writable:=FALSE, 	TPDO_Mappable:=TRUE);
	Max_slippage													: ST_CAN_Object := (Name:='Max slippage', 											Index:=16#60F8,				 								RPDO_Mappable:=TRUE);
	Control_effort													: ST_CAN_Object := (Name:='Control effort', 										Index:=16#60FA,				 			Writable:=FALSE, 	TPDO_Mappable:=TRUE);
	Position_demand_integral_value									: ST_CAN_Object := (Name:='Position demand integral value', 						Index:=16#60FC,				 			Writable:=FALSE, 	TPDO_Mappable:=TRUE);
	Digital_inputs													: ST_CAN_Object := (Name:='Digital inputs', 										Index:=16#60FD,				 			Writable:=FALSE, 	TPDO_Mappable:=TRUE);
	Digital_outputs_Highest_sub_index_supported						: ST_CAN_Object := (Name:='Digital outputs_Highest sub-index supported', 			Index:=16#60FE,				 Length:=1, Writable:=FALSE, 							Default_Value:=2, 	SubElements:=E_SubElement_types.With_fix_subelements);
	Digital_outputs_Physical_outputs								: ST_CAN_Object := (Name:='Digital outputs_Physical outputs', 						Index:=16#60FE, Subindex:=1, 								RPDO_Mappable:=TRUE, 						SubElements:=E_SubElement_types.Fix_subelement);
	Digital_outputs_bit_mask										: ST_CAN_Object := (Name:='Digital outputs_Bit mask',			 					Index:=16#60FE, Subindex:=2, 								RPDO_Mappable:=TRUE, 						SubElements:=E_SubElement_types.Fix_subelement);
	Target_velocity													: ST_CAN_Object := (Name:='Target velocity', 										Index:=16#60FF,				 								RPDO_Mappable:=TRUE);
	
	// Motor data
	Motor_type														: ST_CAN_Object := (Name:='Motor type', 											Index:=16#6402,				 Length:=2);
	Motor_catalogue_number											: ST_CAN_Object := (Name:='Motor catalogue number', 								Index:=16#6403,				 Length:=0);
	Motor_manufacturer												: ST_CAN_Object := (Name:='Motor manufacturer', 									Index:=16#6404,				 Length:=0);
	http_motor_catalogue_address									: ST_CAN_Object := (Name:='http motor catalogue address', 							Index:=16#6405,				 Length:=0);
	Supported_drive_modes											: ST_CAN_Object := (Name:='Supported drive modes', 									Index:=16#6502,				 			Writable:=FALSE,	TPDO_Mappable:=TRUE);
	Drive_catalogue_number											: ST_CAN_Object := (Name:='Drive catalogue number', 								Index:=16#6503,				 Length:=0);
	http_drive_catalogue_address									: ST_CAN_Object := (Name:='http drive catalogue address', 							Index:=16#6505,				 Length:=0);	
	Version_number													: ST_CAN_Object := (Name:='Version number', 										Index:=16#67FE,				 			Writable:=FALSE);
	Single_device_type												: ST_CAN_Object := (Name:='Single device type', 									Index:=16#67FF,				 			Writable:=FALSE);	
END_VAR

// ---- GVLs/GLB.TcGVL
{attribute 'qualified_only'}
VAR_GLOBAL
	Logger			: FB_Logger;
	ADSNetID_CAN	: STRING(23) := '5.156.6.243.3.1';	// ADSNETID of the CAN module
	NodeID			: BYTE :=2;								// Node ID of the controller	
END_VAR

// ---- GVLs/Manufacturer_Label_Objects.TcGVL
{attribute 'qualified_only'}
VAR_GLOBAL
	Serial_Number			: ST_CAN_Object := (Name:='Serial Number', 			Index:=16#41C0, Subindex:=16#01);
	Model_Info				: ST_CAN_Object := (Name:='Model Info', 			Index:=16#41C0, Subindex:=16#02, Length:=255);
	Min_v					: ST_CAN_Object := (Name:='Min v', 					Index:=16#41C0, Subindex:=16#03);
	Max_v					: ST_CAN_Object := (Name:='Max v', 					Index:=16#41C0, Subindex:=16#04);
	Motor_rated_current		: ST_CAN_Object := (Name:='Motor rated current', 	Index:=16#41C0, Subindex:=16#05);
	Drive_rated_current		: ST_CAN_Object := (Name:='Drive rated current', 	Index:=16#41C0, Subindex:=16#06);
	Max_current				: ST_CAN_Object := (Name:='Max current', 			Index:=16#41C0, Subindex:=16#07, Length:=2);
	Motor_rated_torque		: ST_CAN_Object := (Name:='Motor rated torque', 	Index:=16#41C0, Subindex:=16#08);
	Max_torque				: ST_CAN_Object := (Name:='Max torque', 			Index:=16#41C0, Subindex:=16#09, Length:=2);
	Motor_rated_speed		: ST_CAN_Object := (Name:='Motor rated speed', 		Index:=16#41C0, Subindex:=16#0A);
	Number_of_pole_pairs	: ST_CAN_Object := (Name:='Number of pole pairs', 	Index:=16#41C0, Subindex:=16#0B, Length:=2);
	Motor_torque_constant	: ST_CAN_Object := (Name:='Motor torque constant', 	Index:=16#41C0, Subindex:=16#0C);
	Flux_producing_P_gain	: ST_CAN_Object := (Name:='Flux producing P gain', 	Index:=16#41C0, Subindex:=16#0D);
	Flux_producing_I_gain	: ST_CAN_Object := (Name:='Flux producing I gain', 	Index:=16#41C0, Subindex:=16#0E);
	Torque_producing_P_ain	: ST_CAN_Object := (Name:='Torque producing P ain', Index:=16#41C0, Subindex:=16#0F);
	Torque_producing_I_gain	: ST_CAN_Object := (Name:='Torque producing I gain',Index:=16#41C0, Subindex:=16#10);
	Magnetic_encoder_offset	: ST_CAN_Object := (Name:='Magnetic encoder offset',Index:=16#41C0, Subindex:=16#11, Length:=2);
	Motor_with_brake		: ST_CAN_Object := (Name:='Motor with brake', 		Index:=16#41C0, Subindex:=16#12, Length:=2);
	Encoder_mode_adjust		: ST_CAN_Object := (Name:='Encoder mode adjust', 	Index:=16#41C0, Subindex:=16#13, Length:=2);
	Motor_max_speed			: ST_CAN_Object := (Name:='Motor max speed', 		Index:=16#41C0, Subindex:=16#14, Length:=2);
	Rotor_inertia			: ST_CAN_Object := (Name:='Rotor inertia', 			Index:=16#41C0, Subindex:=16#15);
	Motor_Time_At_Peak		: ST_CAN_Object := (Name:='Motor Time At Peak', 	Index:=16#41C0, Subindex:=16#17);
	Drive_Time_At_Peak		: ST_CAN_Object := (Name:='Drive Time At Peak', 	Index:=16#41C0, Subindex:=16#18);
	Single_Turn_Resolution	: ST_CAN_Object := (Name:='Single-Turn Resolution', Index:=16#41C0, Subindex:=16#19, Length:=1);
	Multi_Turn_Resolution	: ST_CAN_Object := (Name:='Multi Turn Resolution', 	Index:=16#41C0, Subindex:=16#1A, Length:=1);

	Manufacturer_Label_Objects_List : ARRAY [0..24] OF ST_CAN_Object := [Serial_Number, Model_Info, Min_v, Max_v, Motor_rated_current, Drive_rated_current, Max_current, Motor_rated_torque, Max_torque, Motor_rated_speed, Number_of_pole_pairs, Motor_torque_constant, Flux_producing_P_gain, Flux_producing_I_gain, Torque_producing_P_ain, Torque_producing_I_gain, Magnetic_encoder_offset, Motor_with_brake, Encoder_mode_adjust, Motor_max_speed, Rotor_inertia, Motor_Time_At_Peak, Drive_Time_At_Peak, Single_Turn_Resolution, Multi_Turn_Resolution];
END_VAR

// ---- GVLs/Manufacturer_specific_Object_List.TcGVL
{attribute 'qualified_only'}
VAR_GLOBAL
	Current_Offset_Feedback_NrOfObjects	: ST_CAN_Object	:= (Name:='Current Offset Feedback_NrOfObjects',	Index:=16#2005, 				Length:=1,	Default_Value:=3);
	Current_Offset_Feedback_Phase_A		: ST_CAN_Object	:= (Name:='Current Offset Feedback_Phase A', 		Index:=16#2005,	Subindex:=1);
	Current_Offset_Feedback_Phase_B		: ST_CAN_Object	:= (Name:='Current Offset Feedback_Phase B', 		Index:=16#2005,	Subindex:=2);
	Current_Offset_Feedback_Phase_C		: ST_CAN_Object	:= (Name:='Current Offset Feedback_Phase C', 		Index:=16#2005,	Subindex:=3);
	VF_Commutation_Frequency			: ST_CAN_Object := (Name:='VF Commutation Frequency', 				Index:=16#2008, 												Default_Value:=5);
	Motor_Feedback_Current_NrOfObjects	: ST_CAN_Object := (Name:='Motor Feedback Current_NrOfObjects', 	Index:=16#2020,					Length:=1, 	Default_Value:=3);
	Motor_Feedback_Current_Phase_A		: ST_CAN_Object := (Name:='Motor Feedback Current_Phase A', 		Index:=16#2020,	Subindex:=1);
	Motor_Feedback_Current_Phase_B		: ST_CAN_Object := (Name:='Motor Feedback Current_Phase B', 		Index:=16#2020,	Subindex:=2);
	Motor_Feedback_Current_Phase_C		: ST_CAN_Object := (Name:='Motor Feedback Current_Phase C', 		Index:=16#2020,	Subindex:=3);
	PWM_duty_cycle_NrOfObjects			: ST_CAN_Object := (Name:='PWM duty cycle_NrOfObjects', 			Index:=16#2022,					Length:=1, 	Default_Value:=3);
	PWM_duty_cycle_Phase_A				: ST_CAN_Object := (Name:='PWM duty cycle_Phase A', 				Index:=16#2022,	Subindex:=1);
	PWM_duty_cycle_Phase_B				: ST_CAN_Object := (Name:='PWM duty cycle_Phase B', 				Index:=16#2022,	Subindex:=2);
	PWM_duty_cycle_Phase_C				: ST_CAN_Object := (Name:='PWM duty cycle_Phase C', 				Index:=16#2022,	Subindex:=3);
	Electrical_commutation_Degrees		: ST_CAN_Object := (Name:='Electrical commutation Degrees', 		Index:=16#2025);
	Current_limit						: ST_CAN_Object := (Name:='Current limit', 							Index:=16#2028);
	Peak_current						: ST_CAN_Object := (Name:='Peak current', 							Index:=16#2029, 							Default_Value:=180);
	Continuous_Current					: ST_CAN_Object	:= (Name:='Continuous Current', 					Index:=16#202A, 							Default_Value:=100);
	Direct_axis_NrOfObjects				: ST_CAN_Object := (Name:='Direct axis_NrOfObjects',				Index:=16#2030,					Length:=1, 	Default_Value:=4);
	Direct_axis_Current_Feedback		: ST_CAN_Object := (Name:='Direct axis_Current Feedback', 			Index:=16#2030,	Subindex:=1);
	Direct_axis_Current_Error			: ST_CAN_Object := (Name:='Direct axis_Current Error', 				Index:=16#2030,	Subindex:=2);
	Direct_axis_Reference_current		: ST_CAN_Object := (Name:='Direct axis_Reference current', 			Index:=16#2030,	Subindex:=3);
	Direct_axis_Voltage_demand			: ST_CAN_Object := (Name:='Direct axis_Voltage demand', 			Index:=16#2030,	Subindex:=4);
	Quadrature_axis_NrOfObjects			: ST_CAN_Object := (Name:='Quadrature axis_NrOfObjects', 			Index:=16#2031,					Length:=1, 	Default_Value:=4);
	Quadrature_axis_Current_Feedback	: ST_CAN_Object := (Name:='Quadrature axis_Current Feedback', 		Index:=16#2031,	Subindex:=1);
	Quadrature_axis_Current_Error		: ST_CAN_Object := (Name:='Quadrature axis_Current Error', 			Index:=16#2031,	Subindex:=2);
	Quadrature_axis_Reference_current	: ST_CAN_Object := (Name:='Quadrature axis_Reference current', 		Index:=16#2031,	Subindex:=3);
	Quadrature_axis_Voltage_demand		: ST_CAN_Object := (Name:='Quadrature axis_Voltage demand', 		Index:=16#2031,	Subindex:=4);
	Current_Following_Error_NrOfObjects	: ST_CAN_Object := (Name:='Current Following Error_NrOfObjects', 	Index:=16#2034,					Length:=1, 	Default_Value:=2);
	Current_Following_Error_Window		: ST_CAN_Object := (Name:='Current Following Error_Window', 		Index:=16#2034,	Subindex:=1,	Length:=2, 						Default_Value:=7);
	Current_Following_Error_Time_Out	: ST_CAN_Object := (Name:='Current Following Error_Time Out', 		Index:=16#2034,	Subindex:=2,	Length:=2, 						Default_Value:=8);
	Homing_Block_NrOfObjects			: ST_CAN_Object := (Name:='Homing Block_NrOfObjects', 				Index:=16#2035,					Length:=1, 	Default_Value:=2);
	Homing_Block_Blocking_current		: ST_CAN_Object := (Name:='Homing Block_Blocking current', 			Index:=16#2035,	Subindex:=1,	Length:=2);
	Homing_Block_Blocking_time			: ST_CAN_Object := (Name:='Homing Block_Blocking time', 			Index:=16#2035,	Subindex:=2,	Length:=2);
	I2T_NrOfObjects						: ST_CAN_Object := (Name:='I2T_NrOfObjects', 						Index:=16#2038,					Length:=1, 	Default_Value:=2);
	I2T_Motor_Thermal_Saturation		: ST_CAN_Object := (Name:='I2T_Motor Thermal Saturation', 			Index:=16#2038,	Subindex:=1,	Length:=2);
	I2T_Drive_Thermal_Saturation		: ST_CAN_Object := (Name:='I2T_Drive Thermal Saturation', 			Index:=16#2038,	Subindex:=2,	Length:=2);
	Torque_Feedback						: ST_CAN_Object := (Name:='Torque Feedback', 						Index:=16#2044);
	Velocity_loop_integral_gain			: ST_CAN_Object := (Name:='Velocity loop integral gain', 			Index:=16#2050, 												Default_Value:=5);
	Velocity_loop_proportional_gain		: ST_CAN_Object := (Name:='Velocity loop proportional gain', 		Index:=16#2051, 												Default_Value:=1);
	Velocity_loop_torque_limit			: ST_CAN_Object := (Name:='Velocity loop torque limit', 			Index:=16#2053);
	Velocity_Loop_Advanced_Tuning_Switch: ST_CAN_Object := (Name:='Velocity Loop Advanced Tuning Switch', 	Index:=16#2054,					Length:=2);
	Velocity_Loop_Target_Bandwidth		: ST_CAN_Object := (Name:='Velocity Loop Target Bandwidth', 		Index:=16#2055);
	Velocity_Loop_Damping_Ratio			: ST_CAN_Object := (Name:='Velocity Loop Damping Ratio', 			Index:=16#2056);
	Homing_Velocity_Invert				: ST_CAN_Object := (Name:='Homing Velocity Invert', 				Index:=16#2060,					Length:=2);
	Homing_Time_Out						: ST_CAN_Object := (Name:='Homing Time Out', 						Index:=16#2061,					Length:=2);
	Velocity_Following_Error_NrOfObjects: ST_CAN_Object := (Name:='Velocity Following Error_NrOfObjects', 	Index:=16#2064,					Length:=1, 	Default_Value:=2);
	Velocity_Following_Error_Window		: ST_CAN_Object := (Name:='Velocity Following Error_Window', 		Index:=16#2064,	Subindex:=1,	Length:=2);
	Velocity_Following_Error_Time_Out	: ST_CAN_Object := (Name:='Velocity Following Error_Time Out', 		Index:=16#2064,	Subindex:=2,	Length:=2);
	Average_Feedback_Velocity			: ST_CAN_Object := (Name:='Average Feedback Velocity', 				Index:=16#2070);
	Feedback_Velocity					: ST_CAN_Object := (Name:='Feedback Velocity', 						Index:=16#2071);
	
	// Position
	Encoder_Counts						: ST_CAN_Object := (Name:='Encoder Counts', 						Index:=16#2072);
	SingleTurn_Position					: ST_CAN_Object := (Name:='SingleTurn Position', 					Index:=16#2073, 	TPDO_Mappable:=TRUE,	Default_Value:=0);
	MultiTurn_Position					: ST_CAN_Object := (Name:='MultiTurn Position', 					Index:=16#2074, 	TPDO_Mappable:=TRUE,	Default_Value:=0);
	
	J_Observer_Curve_Type				: ST_CAN_Object := (Name:='J Observer Curve Type', 					Index:=16#2080,					Length:=1);
	J_Observer_Cycle_No					: ST_CAN_Object := (Name:='J Observer Cycle No', 					Index:=16#2081,					Length:=1);
	J_Observer_Max_Speed				: ST_CAN_Object := (Name:='J Observer Max Speed', 					Index:=16#2082,					Length:=2);
	J_Observer_Max_Speed_Time			: ST_CAN_Object := (Name:='J Observer Max Speed Time', 				Index:=16#2083,					Length:=2);
	J_Observer_Zero_Speed_Time			: ST_CAN_Object := (Name:='J Observer Zero Speed Time', 			Index:=16#2084,					Length:=2);
	J_Observer_Acceleration_Rate		: ST_CAN_Object := (Name:='J Observer Acceleration Rate', 			Index:=16#2085,					Length:=2);
	J_Observer_Deceleration_Rate		: ST_CAN_Object := (Name:='J Observer Deceleration Rate', 			Index:=16#2086,					Length:=2);
	J_Observer_Speed_Limit_High			: ST_CAN_Object := (Name:='J Observer Speed Limit High', 			Index:=16#2087,					Length:=2);
	J_Observer_Speed_Limit_Low			: ST_CAN_Object := (Name:='J Observer Speed Limit Low', 			Index:=16#2088,					Length:=2);
	Position_loop_proportional_gain		: ST_CAN_Object := (Name:='Position loop proportional gain', 		Index:=16#20A1,								Default_Value:=25);
	Home_Position						: ST_CAN_Object := (Name:='Home Position', 							Index:=16#20C0);
	Total_inertia						: ST_CAN_Object := (Name:='Total inertia', 							Index:=16#2102);
	Enable_Field_Weakening				: ST_CAN_Object := (Name:='Enable Field Weakening', 				Index:=16#2104,					Length:=2);
	Invert_feedback_direction			: ST_CAN_Object := (Name:='Invert feedback direction', 				Index:=16#2107,					Length:=2);
	Field_Weakening_Max					: ST_CAN_Object := (Name:='Field Weakening Max', 					Index:=16#2108);
	Field_Weakening_Threshold			: ST_CAN_Object := (Name:='Field Weakening Threshold', 				Index:=16#2109);
	Field_Weakening_Gain				: ST_CAN_Object := (Name:='Field Weakening Gain', 					Index:=16#210A);
	Drive_operating_mode				: ST_CAN_Object := (Name:='Drive operating mode', 					Index:=16#2140,					Length:=2);
	
	// Brake
	Brake_NrOfObjects					: ST_CAN_Object := (Name:='Brake_NrOfObjects', 						Index:=16#2150,					Length:=1,	Default_Value:=4);
	Brake_Status						: ST_CAN_Object := (Name:='Brake_Status', 							Index:=16#2150,	Subindex:=1,	Length:=2);
	Brake_Override						: ST_CAN_Object := (Name:='Brake_Override', 						Index:=16#2150,	Subindex:=2,	Length:=2);
	Brake_Delay							: ST_CAN_Object := (Name:='Brake_Delay', 							Index:=16#2150,	Subindex:=3);
	Brake_Fault_Delay					: ST_CAN_Object := (Name:='Brake_Fault Delay', 						Index:=16#2150,	Subindex:=4);
	
	Command_Value						: ST_CAN_Object := (Name:='Command Value',							Index:=16#2170, 							Default_Value:=5);
	
